// TwinCAT 3 PLC project REFLEX_3000_PLC
// ProgramVersion: 3.1.4023.0
// libraries:
//   Festo_HomingLibrary, * (Festo)
//   Festo_PtP_Base, * (Festo)
//   Festo_PtP_CiA402_ETC_CMMT_AS, * (Festo)
//   Festo_PtP_CiA402_ETC_CMMT_ST, * (Festo)
//   Tc2_EtherCAT, * (Beckhoff Automation GmbH)
//   Tc2_MC2, * (Beckhoff Automation GmbH)
//   Tc2_MC2_Drive, * (Beckhoff Automation GmbH)
//   Tc2_ModbusRTU, * (Beckhoff Automation GmbH)
//   Tc2_SerialCom, * (Beckhoff Automation GmbH)
//   Tc2_Standard, * (Beckhoff Automation GmbH)
//   Tc2_System, * (Beckhoff Automation GmbH)
//   Tc2_Utilities, * (Beckhoff Automation GmbH)
//   Tc3_EventLogger, * (Beckhoff Automation GmbH)
//   Tc3_Mc3Definitions, * (Beckhoff Automation GmbH)
//   Tc3_McCollisionAvoidance, * (Beckhoff Automation GmbH)
//   Tc3_McCoordinatedMotion, * (Beckhoff Automation GmbH)
//   Tc3_Module, * (Beckhoff Automation GmbH)
//   Util, * (System)
//   Tc3_XTS_Utility,3.1.2202.3,Beckhoff Automation GmbH
// project tree:
//   DUTs/ Running_Recipe.TcDUT
//   FB/Keyence_Laser/ FB_Keyence_Laser_Steuerung.TcPOU, ST_KeyenceLaser_Completion_Status.TcDUT, ST_KeyenceLaser_Count_Result_Data.TcDUT, ST_KeyenceLaser_ErrorStatus.TcDUT, ST_KeyenceLaser_Error_Codes.TcDUT, ST_KeyenceLaser_Function_Request.TcDUT, ST_KeyenceLaser_Function_Status.TcDUT, ST_KeyenceLaser_General_Request.TcDUT, ST_KeyenceLaser_Machine_Status.TcDUT, ST_KeyenceLaser_Operate_Parameter.TcDUT, ST_KeyenceLaser_Request_Completion_Clear.TcDUT, ST_KeyenceLaser_TwoD_Code_Read_Result.TcDUT
//   FB/Keyence_Laser/ST_Keyence/Input/ ST_KeyenceLaser_Block_Edit_Request_Completion_Status.TcDUT, ST_KeyenceLaser_Block_Edit_Request_Error_Status.TcDUT, ST_KeyenceLaser_Command_Request_Completion_Status.TcDUT, ST_KeyenceLaser_Command_Request_Error.TcDUT, ST_KeyenceLaser_Control_Status.TcDUT, ST_KeyenceLaser_Edit_Request_Completion_Status.TcDUT, ST_KeyenceLaser_Edit_Request_Error_Status.TcDUT, ST_KeyenceLaser_Function_Status_I.TcDUT, ST_KeyenceLaser_General_Request_Completion_Status.TcDUT, ST_KeyenceLaser_General_Request_Error_Status.TcDUT, ST_KeyenceLaser_General_Status.TcDUT, ST_KeyenceLaser_IO_Status.TcDUT, ST_KeyenceLaser_Operation_Request_Completion_Status.TcDUT, ST_KeyenceLaser_Operation_Request_Error_Status.TcDUT, ST_KeyenceLaser_Running_Status.TcDUT
//   FB/Keyence_Laser/ST_Keyence/Output/ ST_KeyenceLaser_Block_Edit_Request.TcDUT, ST_KeyenceLaser_Block_Edit_Request_Completion_Clear.TcDUT, ST_KeyenceLaser_Command_Request.TcDUT, ST_KeyenceLaser_Command_Request_Completion_Clear.TcDUT, ST_KeyenceLaser_Edit_Request.TcDUT, ST_KeyenceLaser_Edit_Request_Completion_Clear.TcDUT, ST_KeyenceLaser_Function_Request_I.TcDUT, ST_KeyenceLaser_General_Request_Completion_Clear.TcDUT, ST_KeyenceLaser_General_Request_I.TcDUT, ST_KeyenceLaser_Operating_Request.TcDUT, ST_KeyenceLaser_Operating_Request_Completion_Clear.TcDUT
//   FB/ OP10_ROBO_PNP.TcPOU, Servo_Conveyor_FB_OP90.TcPOU, Cylinder_Block.TcPOU, Cylinder_Block_FOR_OP130.TcPOU, Cylinder_Block_HOMING.TcPOU, FB_cycleTime.TcPOU, FB_SimClock.TcPOU, In_Range.TcPOU, Mode_Selection_Block1.TcPOU, OP10_ORING_PNP.TcPOU, OP140_LeakTesting.TcPOU, Pulse_1s.TcPOU, Servo_Conveyor_FB.TcPOU, TestSeq.TcPOU
//   FB/tool/ step_cycle_time.TcPOU, tool_changeover.TcPOU
//   POU1/ FB_Time_Stamp_Maddy.TcPOU, Axis_Position_Bias.TcPOU, MAIN.TcPOU, Recipe_Values.TcGVL, RFID.TcPOU
//   POUs/Programs/OP10/ Body_Singulation_Seq.TcPOU, OP10A_AUTO.TcPOU, OP10A_Camera_FB.TcPOU, OP10A_Conveyor_Prog.TcPOU, OP10A_OP10B_DRUM_FEEDER.TcPOU, OP10B_AUTO.TcPOU, OP10B_Camera_FB.TcPOU, OP10B_Conveyor_Prog.TcPOU, OP10_AUTO.TcPOU, OP10_Body_Camera_Seq.TcPOU, OP10_HMI_GVL.TcGVL, OP10_HOMING.TcPOU, OP10_MAIN.TcPOU, OP10_MANUAL.TcPOU, OP10_ROBO.TcPOU, OP10_SERVO.TcPOU, OP10_VARIABLE.TcGVL
//   POUs/Programs/OP120/ Bypass.TcDUT, OP120_AutoSequence.TcPOU, op120_camera_FB.TcPOU, OP120_Error.TcPOU, OP120_Feed_Conveyor.TcPOU, OP120_GVL.TcGVL, OP120_Initialization_Seq.TcPOU, OP120_IO_Tag_Link.TcGVL, OP120_LockInsert_AutoSequence.TcPOU, OP120_Main.TcPOU, OP120_Manual.TcPOU, OP120_Recipe.TcDUT, OP120_Robo_Byte_Mapping.TcPOU, OP120_Robo_Inputs.TcPOU, OP120_Sing_Auto_PRG.TcPOU
//   POUs/Programs/OP130/ op130_tool_change.TcPOU, OP130_AutoSequence.TcPOU, OP130_Error.TcPOU, OP130_GVL.TcGVL, OP130_Initialization_Seq.TcPOU, OP130_LH_Auto.TcPOU, OP130_Main.TcPOU, OP130_Manual.TcPOU, OP130_Recipe.TcDUT, OP130_RH_Auto.TcPOU, OP130_RH_Initialization_Seq.TcPOU
//   POUs/Programs/OP140/ op140_tool_change.TcPOU, Ateq_Comm_Prog.TcPOU, op140_ateq_fb.TcPOU, OP140_AutoSequence_1.TcPOU, OP140_AutoSequence_2.TcPOU, OP140_AutoSequence_3.TcPOU, OP140_Error.TcPOU, OP140_GVL.TcGVL, OP140_HMI_GVL.TcGVL, OP140_Initialization_Seq.TcPOU, OP140_Main.TcPOU, OP140_Manual.TcPOU
//   POUs/Programs/OP150/ OP150_B.TcPOU, OP150_Laser_FB.TcPOU, Rejection_Codes_Function.TcPOU, OP150_A.TcPOU, OP150_C.TcPOU, OP150_GVL.TcGVL, OP150_Main.TcPOU
//   POUs/Programs/OP20/ OP20_AUTOSEQUENCE.TcPOU, OP20_ERROR.TcPOU, OP20_GVL.TcGVL, OP20_Initialization_Seq.TcPOU, OP20_MAIN.TcPOU, OP20_MANUAL.TcPOU, OP20_Recipe.TcGVL
//   POUs/Programs/OP30/ OP30_Camera_FB.TcPOU, OP30_Conveyor_Cam_Seq.TcPOU, Camera_Job_Change.TcPOU, OP30_AUTOSEQUENCE.TcPOU, OP30_Error.TcPOU, OP30_GVL.TcGVL, OP30_HMI_TAGS.TcGVL, OP30_Initialize_Seq.TcPOU, OP30_MAIN.TcPOU, OP30_MANUAL.TcPOU, OP30_Recipe.TcGVL
//   POUs/Programs/OP40/ op40_toolchangeover.TcPOU, OP40_AUTOSEQUENCE.TcPOU, OP40_ERROR.TcPOU, OP40_GVL.TcGVL, OP40_Initialization_Seq.TcPOU, OP40_MAIN.TcPOU, OP40_MANUAL.TcPOU, OP40_Recipe.TcGVL
//   POUs/Programs/OP50/ OP50_Camera_FB.TcPOU, OP50_Conveyor_Cam_Seq.TcPOU, OP50_AUTOSEQUENCE.TcPOU, OP50_CONVEYOR.TcPOU, OP50_Error.TcPOU, OP50_GVL.TcGVL, OP50_HMI_GVL.TcGVL, OP50_Initialize_Seq.TcPOU, OP50_MAIN.TcPOU, OP50_MANUAL.TcPOU, OP50_Recipe.TcGVL
//   POUs/Programs/OP60/ op60_toolchangeover.TcPOU, OP60_AUTOSEQUENCE.TcPOU, OP60_ERROR.TcPOU, OP60_GVL.TcGVL, OP60_Initialization_Seq.TcPOU, OP60_MAIN.TcPOU, OP60_MANUAL.TcPOU, OP60_Recipe.TcGVL
//   POUs/Programs/OP70/ OP70_Camera_FB.TcPOU, OP70_Conveyor_Cam_Seq.TcPOU, OP70_AUTOSEQUENCE.TcPOU, OP70_CONVEYOR.TcPOU, OP70_Error.TcPOU, OP70_GVL.TcGVL, OP70_Initialize_Seq.TcPOU, OP70_MAIN.TcPOU, OP70_MANUAL.TcPOU, OP70_Recipe.TcGVL
//   POUs/Programs/OP80/ op80_toolchangeover.TcPOU, OP80_AUTOSEQUENCE.TcPOU, OP80_ERROR.TcPOU, OP80_GVL.TcGVL, OP80_HMI_GVL.TcGVL, OP80_Initialization_Seq.TcPOU, OP80_MAIN.TcPOU, OP80_MANUAL.TcPOU, OP80_Recipe.TcGVL
//   POUs/Programs/OP90/ OP90_Camera_Fb.TcPOU, OP90_AUTO.TcPOU, OP90_CAMERA.TcPOU, OP90_Conveyor_FBs.TcPOU, OP90_HMI_GVL.TcGVL, OP90_HOMING.TcPOU, OP90_MAIN.TcPOU, OP90_MANUAL.TcPOU, OP90_SERVO.TcPOU, OP90_VARIABLE.TcGVL
//   POUs/Programs/XTS/ Fb_MoverSequence.TcPOU, HMI_GVL.TcGVL, MAIN_1.TcPOU, PRG_XTS_Sequence.TcPOU, XTS_GVL.TcGVL
//   / Robot_Comm_Task.TcTTO, PlcTask.TcTTO, RecipeManager.TcRMO (not stored)
//   DUTs/OP10/ OP10_GRP_CONTRL.TcDUT, OP10_GRP_STATUS.TcDUT, OP10_ORNG_CYL_DLY.TcDUT, OP10_ORNG_CYL_IP.TcDUT, OP10_ORNG_CYL_OP.TcDUT, OP10_ROBO_CNTRL.TcDUT, OP10_ROBO_STUS.TcDUT
//   DUTs/XTS/ STATION_DONE.TcDUT
//   FB/Axis/ ENUM_Axis.TcDUT, FB_Axis.TcPOU, FB_Axis_FESTO.TcPOU, OP10_SERVO_LIMIT.TcDUT, OP90_SERVO_LIMIT.TcDUT, Servo_Control.TcDUT, stManualModeAxis.TcDUT
//   FB/Cognex_Camera/ Acquisition_control.TcDUT, Acquisition_status.TcDUT, FB_Cognex_ProfiNET_1.TcPOU, Inspection_control.TcDUT, Inspection_status.TcDUT, UNION_64Byte.TcDUT
//   FB/FB/FB/ ATEQ_LEAK.TcPOU
//   FB/RFID/ FB_RFID.TcPOU, Head1.TcDUT, HeadData.TcDUT, Memory.TcDUT, UNION_RFID.TcDUT
//   FB/Robot/ E_State_RobotGeneral.TcDUT, FB_Robot.TcPOU
//   FB/Scanner/ Acquisition_Control_Scanner.TcDUT, Acquisition_Status_Scanner.TcDUT, Result_Control_Scanner.TcDUT, Result_Data_Register.TcDUT, Result_Status.TcDUT, Scanner.TcPOU
//   FB/Schunk/ ENUM_Schunk.TcDUT, FB_Schunk.TcPOU, FC_Real_Convert.TcPOU, iSchunkProcessData.TcDUT, oSchunkProcessData.TcDUT, stManualModeAxis_1.TcDUT, UNION_iSchunkProcessData.TcDUT, UNION_oSchunkProcessData.TcDUT, UNION_REAL.TcDUT
//   GVLs/ E_EcCommState.TcDUT, GVL.TcGVL, RayPRO_Variables.TcGVL, SerialComm.TcGVL, ST_SlaveState.TcDUT, ST_SlaveStateInfo.TcDUT (not stored)
//   GVLs/XTS/ GVL_XTS.TcGVL
//   POUs/ Error.TcPOU
//   POUs/GENERAL/ Robot_232_Comm_Prgrm.TcPOU, EtherCatDiag.TcPOU, GENERAL_VARIABLE.TcGVL, IO_Diag.TcPOU, MODE_SELECTION.TcPOU
//   POUs/IO/ OP120_JB_IO.TcPOU, OP160_MASTER4_IO.TcPOU, OP160_MP_IO.TcPOU, OP90_JB_IO.TcPOU, OP90_MASTER3_IO.TcPOU, OP90_MP_IO.TcPOU
//   POUs/IO_GVLs/ Master3_IO.TcGVL, Master4_IO.TcGVL, OP120_JB.TcGVL, OP160_MP.TcGVL, OP90_JB.TcGVL, OP90_MP.TcGVL, SAFETY_IOs.TcGVL
//   POUs/IO_Mapping_OP10JB/ IO_OP10A_10B_JB.TcPOU, IO_OP10_JB_IO.TcGVL
//   POUs/IO_mapping_OP10MP/ IO_OP10_MP.TcGVL, IO_OP10_PANEL.TcPOU
//   POUs/OP10_Profinet_IO/ Master1_IO.TcGVL, Master1_IO_Map.TcPOU, MASTER2_IO.TcGVL, MASTER2_IO_Map.TcPOU
//   POUs/Programs/ Error_GVL.TcGVL
//   POUs/Programs/offline testing/ cylinder_2_pos.TcPOU, cylinder_3_pos.TcPOU, Cylinder_Block_v1.TcPOU, cylinder_validation_st.TcPOU, offline_fb.TcPOU, offline_main.TcPOU, POU_1.TcPOU, servo.TcPOU, servo_validation.TcPOU
//   POUs/Programs/OP10A_Bowl/ Bowl_Control.TcPOU
//   POUs/Programs/OP110/ OP110_AUTOSEQUENCE.TcPOU, OP110_ERROR.TcPOU, OP110_GVL.TcGVL, OP110_HMI_GVL.TcGVL, OP110_Initialization_Seq.TcPOU, OP110_MAIN.TcPOU, OP110_MANUAL.TcPOU, OP110_Recipe.TcGVL
//   POUs/Programs/OP160/ OP160_AutoSequence.TcPOU, OP160_Error.TcPOU, OP160_GVL.TcGVL, OP160_Initialization_Seq.TcPOU, OP160_IO_Tag_Link.TcGVL, OP160_Main.TcPOU, OP160_Manual.TcPOU, OP160_QCPlace_AutoSequence.TcPOU, OP160_Recipe.TcDUT, OP160_RFID.TcPOU, OP160_Robo_Byte_Mapping.TcPOU, OP160_Robo_Inputs.TcPOU

CONFIGURATION REFLEX_3000_PLC
    RESOURCE PLC ON TwinCAT3
        TASK Robot_Comm_Task(INTERVAL := T#1ms, PRIORITY := 19);
        TASK PlcTask(INTERVAL := T#10ms, PRIORITY := 20);
        PROGRAM Robot_232_Comm_Prgrm WITH Robot_Comm_Task : Robot_232_Comm_Prgrm;
        PROGRAM MAIN WITH PlcTask : MAIN;
    END_RESOURCE
END_CONFIGURATION

// ---- DUTs/Running_Recipe.TcDUT
TYPE Running_Recipe :
STRUCT
//General
	Model_Dia					: STRING[80];
	Part_Number					: STRING[80];
	Body_Conductivity			: BOOL;
	Comp_Per_Bag 				: INT;
		
//OP10	
	OP10_Cam_Prog_Num			: INT;
	OP10_Robot_Prog_Num			: INT;
	OP10_Gripper_Pos			: REAL;

//OP20
	OP20_Vert_Ser_Pos			: REAL;
	OP20_Oiling_Time			: INT;
	
OP20_Oiling_Range				: REAL;

//OP30
	OP30_Cam_Prog_Num			: INT;
	OP30_Grip_Wrk_Pos			: REAL;
	OP30_Vert_Ser_Pick_Pos		: REAL;
	OP30_Vert_Ser_Place_Pos		: REAL;	
	OP30_Hori_Ser_Pick_Pos		: REAL;
	OP30_Hori_Ser_Place_Pos		: REAL;		

//OP40
	OP40_Vert_Ser_Pos			: REAL;
	OP40_LVDT_Chck_Value		: REAL;

//OP40_LVDT_Tolerance				: REAL;

//OP50
	OP50_Cam_Prog_Num			: INT;
	OP50_Vert_Ser_Pick_Pos		: REAL;
	OP50_Vert_Ser_Place_Pos		: REAL;	
	OP50_Hori_Ser_Pick_Pos		: REAL;
	OP50_Hori_Ser_Place_Pos		: REAL;		

//OP60
	OP60_Vert_Ser_Pos			: REAL;
	OP60_LVDT_Chck_Value		: REAL;

//OP60_LVDT_Tolerance				: REAL;

//OP70
	OP70_Cam_Prog_Num			: INT;
	OP70_Grip_Wrk_Pos			: REAL;
	OP70_Vert_Ser_Pick_Pos		: REAL;
	OP70_Vert_Ser_Place_Pos		: REAL;	
	OP70_Hori_Ser_Pick_Pos		: REAL;
	OP70_Hori_Ser_Place_Pos		: REAL;		


//OP80
	OP80_Vert_Ser_Pos			: REAL;
	OP80_LVDT_Chck_Value		: REAL;

//OP80_LVDT_Tolerance				: REAL;

//OP90
	OP90_Cam_Prog_Num			: INT;
	OP90_Vert_Ser_Pick_Pos		: REAL;
	OP90_Vert_Ser_Place_Pos		: REAL;	
	OP90_Hori_Ser_Pick_Pos		: REAL;
	OP90_Hori_Ser_Place_Pos		: REAL;	

//OP110
	OP110_Vert_Ser_Pos			: REAL;
	OP110_Oiling_Time			: INT;
	
OP110_Oiling_Range				: REAL;

//OP120
	OP120_Cam_Prog_Num			: INT;
                            	
//OP130                     	
	OP130_Trq_value				: REAL;
	OP130_Vert_Ser_Pos			: REAL;
	                        	
//OP140                     	
	OP140_Vert_Ser_Pos			: REAL;
	                        	
OP140_Wiping_Cycle				: INT;
OP140_NOK_Retry_Cycle			: INT;
                            	
//OP150-A                   	
	OP150A_Cam_Prog_Num			: INT;
	                        	
//OP150-B                   	
	OP150B_Lsr_Mrk_Job_num		: INT;
	
//OP160
	OP160_Robo_Prog_Num			: INT;	
END_STRUCT
END_TYPE

// ---- FB/Keyence_Laser/ST_KeyenceLaser_Completion_Status.TcDUT
TYPE ST_KeyenceLaser_Completion_Status :
STRUCT
Marking_Complete				: BIT ;
Guide_Laser_Complete			: BIT ;
Laser_Stop_Complete				: BIT ;
Error_Clear_Complete			: BIT ;
TWODC_Read_Complete				: BIT ;
Reserve_15						: BIT ;
Reserve_16						: BIT ;
Reserve_17						: BIT ;
//
PROGRAM_Edit_Complete			: BIT ;
Reserve_18						: BIT ;
Reserve_19						: BIT ;
Reserve_20						: BIT ;
Reserve_21						: BIT ;
Reserve_22						: BIT ;
Reserve_23						: BIT ;
Reserve_24						: BIT ;
//
PROGRAM_Change_Complete			: BIT ;
Rank_Change_Complete			: BIT ;
Counter_No_Complete				: BIT ;
Counter_Value_Complete			: BIT ;
Counter_Up_Complete				: BIT ;
Counter_Down_Complete			: BIT ;
Counter_Reset_Complete			: BIT ;
Reserve_25						: BIT ;
//
ReserveByte_2					: Byte ;
//
Setting_STRING_Read_Complete	: BIT ;
Marked_STRING_Read_Complete		: BIT ;
STRING_Change_Complete			: BIT ;
Reserve_26						: BIT ;
Reserve_27						: BIT ;
Reserve_28						: BIT ;
Reserve_29						: BIT ;
Reserve_30						: BIT ;
//
ReserveWord_2a					: BYTE ;
//
ReserveWord_2b					: BYTE ;
//
Command_Send_Complete			: BIT ;
Reserve_31						: BIT ;
Reserve_32						: BIT ;
Reserve_33						: BIT ;
Reserve_34						: BIT ;
Reserve_35						: BIT ;
Reserve_36						: BIT ;
Reserve_37						: BIT ;
END_STRUCT
END_TYPE

// ---- FB/Keyence_Laser/ST_KeyenceLaser_Count_Result_Data.TcDUT
TYPE ST_KeyenceLaser_Count_Result_Data :
STRUCT
END_STRUCT
END_TYPE

// ---- FB/Keyence_Laser/ST_KeyenceLaser_ErrorStatus.TcDUT
TYPE ST_KeyenceLaser_ErrorStatus :
STRUCT
Start_Marking_Request_Error			: BIT ;
Guide_Laser_Request_Error			: BIT ;
Stop_Marking_Request_Error			: BIT ;
Error_Clear_Request_Error			: BIT ;
TwoDC_Read_Request_Error			: BIT ;//2DC_Read_Request_Error
Reserve_38							: BIT ;
Reserve_39							: BIT ;
Reserve_40							: BIT ;
//
PROGRAM_Edit_Error					: BIT ;
Reserve_41							: BIT ;
Reserve_42							: BIT ;
Reserve_43							: BIT ;
Reserve_44							: BIT ;
Reserve_45							: BIT ;
Reserve_46							: BIT ;
Reserve_47							: BIT ;
//
PROGRAM_Change_Request_Error		: BIT ;
Rank_Change_Request_Error			: BIT ;
Counter_No_Change_Request_Error		: BIT ;
Counter_Value_Change_Request_Error	: BIT ;
Counter_Up_Request_Error			: BIT ;
Counter_Down_Request_Error			: BIT ;
Counter_Reset_Request_Error			: BIT ;
Reserve_48							: BIT ;
//
ReserveByte_3						: Byte ;
//
Setting_STRING_Read_Request_Error	: BIT ;
Marked_STRING_Read_Request_Error	: BIT ;
STRING_Change_Request_Error			: BIT ;
Reserve_49							: BIT ;
Reserve_50							: BIT ;
Reserve_51							: BIT ;
Reserve_52							: BIT ;
Reserve_53							: BIT ;
//
ReserveWord_3a						: Byte ;
//
ReserveWord_3b						: Byte ;
//
Command_Send_Request_Error			: BIT ;
Reserve_54							: BIT ;
Reserve_55							: BIT ;
Reserve_56							: BIT ;
Reserve_57							: BIT ;
Reserve_58							: BIT ;
Reserve_59							: BIT ;
Reserve_60							: BIT ;
END_STRUCT
END_TYPE

// ---- FB/Keyence_Laser/ST_KeyenceLaser_Error_Codes.TcDUT
TYPE ST_KeyenceLaser_Error_Codes :
STRUCT
Error_Code_1				: WORD ;
Error_Code_2				: WORD ;
Command_Send_Error_Status	: WORD ;
ReserveWord_4				: WORD ;
END_STRUCT
END_TYPE

// ---- FB/Keyence_Laser/ST_KeyenceLaser_Function_Request.TcDUT
TYPE ST_KeyenceLaser_Function_Request :
STRUCT
Trigger_Lock_Request	: BIT ;
Operation_Stop_Request	: BIT ;
Laser_Stop_Request		: BIT ;
Date_Hold_Request		: BIT ;
A_Reserve_24			: BIT ;
A_Reserve_25			: BIT ;
A_Reserve_26			: BIT ;
A_Reserve_27			: BIT ;
//
A_ReserveByte_4			: Byte ;
A_ReserveWord1			: Word ;
END_STRUCT
END_TYPE

// ---- FB/Keyence_Laser/ST_KeyenceLaser_Function_Status.TcDUT
TYPE ST_KeyenceLaser_Function_Status :
STRUCT
Trigger_Lock_Status				: BIT ;
Operation_Stop_Status			: BIT ;
Laser_Control_Status			: BIT ;
DATE_Hold_Status				: BIT ;
Reserve_10						: BIT ;
Reserve_11						: BIT ;
Reserve_12						: BIT ;
Reserve_13						: BIT ;
//
DATE_Attach_Status				: BIT ;
Counter_End1_Status				: BIT ;
Counter_End2_Status				: BIT ;
Counter_End3_Status				: BIT ;
Counter_End4_Status				: BIT ;
Mark_Check_TwoDC_Read_OK_Status	: BIT ;//Mark_Check_2DC_Read_OK_Status
Mark_Check_TwoDC_Read_NG_Status	: BIT ;//Mark_Check_2DC_Read_NG_Status
Reserve_14						: BIT ;
//
ReserveWord_1					: WORD ;
END_STRUCT
END_TYPE

// ---- FB/Keyence_Laser/ST_KeyenceLaser_General_Request.TcDUT
TYPE ST_KeyenceLaser_General_Request :
STRUCT
Start_Marking_Request			: BIT ;
Guide_Laser_Request				: BIT ;
Stop_Marking_Request			: BIT ;
Error_Clear_Request				: BIT ;
TwoD_C_Read_Request				: BIT ;//2DC_Read_Request
A_Reserve_1						: BIT ;
A_Reserve_2						: BIT ;
A_Reserve_3						: BIT ;
//
Program_Edit_Start_Request		: BIT ;
A_Reserve_4						: BIT ;
A_Reserve_5						: BIT ;
A_Reserve_6						: BIT ;
A_Reserve_7						: BIT ;
A_Reserve_8						: BIT ;
A_Reserve_9						: BIT ;
A_Reserve_10					: BIT ;
//
Program_Change_Request			: BIT ;
Rank_Change_Request				: BIT ;
Counter_No_Change_Request		: BIT ;
Counter_Value_Change_Request	: BIT ;
Counter_Up_Request				: BIT ;
Counter_Down_Request			: BIT ;
Counter_Reset_Request			: BIT ;
A_Reserve_11					: BIT ;
//
A_ReserveByte_1					: BYTE ;
//
A_ReserveByte_2					: BYTE ;
//
Setting_String_Read_Request		: BIT ;
Marked_String_Read_Request		: BIT ;
STRING_Change_Request			: BIT ;
A_Reserve_12					: BIT ;
A_Reserve_13					: BIT ;
A_Reserve_14					: BIT ;
A_Reserve_15					: BIT ;
A_Reserve_16					: BIT ;
//
A_ReserveByte_3					: Byte ;
//
Command_Send_Request			: BIT ;
A_Reserve_17					: BIT ;
A_Reserve_18					: BIT ;
A_Reserve_19					: BIT ;
A_Reserve_20					: BIT ;
A_Reserve_21					: BIT ;
A_Reserve_22					: BIT ;
A_Reserve_23					: BIT ;
END_STRUCT
END_TYPE

// ---- FB/Keyence_Laser/ST_KeyenceLaser_Machine_Status.TcDUT
TYPE ST_KeyenceLaser_Machine_Status :
STRUCT
Ready_Status						: BIT ;
Error_Status						: BIT ;
Warning_Status						: BIT ;
Error_Warning_Status				: BIT ;
Shutter_Status						: BIT ;
Network_Status						: BIT ;
Reserve_1							: BIT ;
Reserve_2							: BIT ;
//
Laser_Emitted_Status				: BIT ;
Shutter_Control_Status				: BIT ;
Remote_Interlock_Status				: BIT ;
Contacter_Status					: BIT ;
Reserve_3							: BIT ;
Reserve_4							: BIT ;
Reserve_5							: BIT ;
Reserve_6							: BIT ;
//
Busy_Status							: BIT ;
Marking_Busy_Status					: BIT ;
Guide_Laser_Busy_Status				: BIT ;
PROGRAM_Change_Busy_Status			: BIT ;
Communication_Prioirty_Error_Status	: BIT ;
PROGRAM_Edit_Busy_Status			: BIT ;
Mark_Check_TwoDC_Read_Busy_Status	: BIT ;//Mark_Check_/2DC_Read_Busy_Status
Reserve_7							: BIT ;
//
ReserveByte_1						: BYTE ;
END_STRUCT
END_TYPE

// ---- FB/Keyence_Laser/ST_KeyenceLaser_Operate_Parameter.TcDUT
TYPE ST_KeyenceLaser_Operate_Parameter :
STRUCT
PROGRAM_No_Status		: WORD ;
Counter_No_Status		: WORD ;
Counter_Value_Status	: DWORD ;
Rank_Value_Status		: WORD ;
ReserveWord_5			: WORD ;
ReserveDWord_1			: DWORD ;
END_STRUCT
END_TYPE

// ---- FB/Keyence_Laser/ST_KeyenceLaser_Request_Completion_Clear.TcDUT
TYPE ST_KeyenceLaser_Request_Completion_Clear :
STRUCT
Marking_Complete_BIT_Clear					: BIT ;
Guide_Laser_Complete_Bit_Clear				: BIT ;
Stop_Marking_Complete_Bit_Clear				: BIT ;
Error_Clear_Complete_Bit_Clear				: BIT ;
TwoDC_Read_Complete_Bit_Clear				: BIT ;//2DC_Read_Complete_Bit_Clear	
A_Reserve_28								: BIT ;
A_Reserve_29								: BIT ;
A_Reserve_30								: BIT ;
//
Program_Edit_Complete_Bit_Clear				: BIT ;
A_Reserve_31								: BIT ;
A_Reserve_32								: BIT ;
A_Reserve_33								: BIT ;
A_Reserve_34								: BIT ;
A_Reserve_35								: BIT ;
A_Reserve_36								: BIT ;
A_Reserve_37								: BIT ;
//
Program_Change_Complete_Bit_Clear			: BIT ;
Rank_Change_Complete_Bit_Clear				: BIT ;
Counter_No_Change_Complete_Bit_Clear		: BIT ;
Counter_Value_Change_Complete_Bit_Clear		: BIT ;
Count_Up_Complete_Bit_Clear					: BIT ;
Count_Down_Complete_Bit_Clear				: BIT ;
Counter_Reset_Complete_Bit_Clear			: BIT ;
A_Reserve_38								: BIT ;
//
A_ReserveByte_5								: Byte ;
//
Setting_String_Read_Complete_Bit_Clear		: BIT ;
Marked_String_Read_Complete_Bit_Clear		: BIT ;
String_Change_Complete_Bit_Clear			: BIT ;
A_Reserve_39								: BIT ;
A_Reserve_40								: BIT ;
A_Reserve_41								: BIT ;
A_Reserve_42								: BIT ;
A_Reserve_43								: BIT ;
//
A_ReserveByte_6								: Byte ;
//
A_ReserveByte_7								: Byte ;
//
Command_Send_Complete_Bit_Clear				: BIT ;
A_Reserve_44								: BIT ;
A_Reserve_45								: BIT ;
A_Reserve_46								: BIT ;
A_Reserve_47								: BIT ;
A_Reserve_48								: BIT ;
A_Reserve_49								: BIT ;
A_Reserve_50								: BIT ;
END_STRUCT
END_TYPE

// ---- FB/Keyence_Laser/ST_KeyenceLaser_TwoD_Code_Read_Result.TcDUT

TYPE ST_KeyenceLaser_TwoD_Code_Read_Result :
STRUCT
Marking_Check_Score_TwoDC_Read_Grade_Status		: WORD ;
Check_Count_Status								: WORD ;
ReserveDWord_2									: DWORD ;
END_STRUCT
END_TYPE

// ---- FB/Keyence_Laser/ST_Keyence/Input/ST_KeyenceLaser_Block_Edit_Request_Completion_Status.TcDUT
TYPE ST_KeyenceLaser_Block_Edit_Request_Completion_Status :
STRUCT
Character_String_Setting_Read_Complete			: BIT;
Character_String_Printed_Read_Complete			: BIT;
Character_String_Change_Complete				: BIT;
Reserve_0										: BIT;
Reserve_1										: BIT;
Reserve_2										: BIT;
Reserve_3										: BIT;
Reserve_4										: BIT;
END_STRUCT
END_TYPE

// ---- FB/Keyence_Laser/ST_Keyence/Input/ST_KeyenceLaser_Block_Edit_Request_Error_Status.TcDUT
TYPE ST_KeyenceLaser_Block_Edit_Request_Error_Status :
STRUCT
Character_String_Setting_Read_Error				: BIT;
Character_String_Printed_Read_Error				: BIT;
Character_String_Change_Error					: BIT;
Reserve_0										: BIT;
Reserve_1										: BIT;
Reserve_2										: BIT;
Reserve_3										: BIT;
Reserve_4										: BIT;
END_STRUCT
END_TYPE

// ---- FB/Keyence_Laser/ST_Keyence/Input/ST_KeyenceLaser_Command_Request_Completion_Status.TcDUT
TYPE ST_KeyenceLaser_Command_Request_Completion_Status :
STRUCT
Command_Request_Complete			: BIT;
Reserve_0							: BIT;
Reserve_1							: BIT;
Reserve_2							: BIT;
Reserve_3							: BIT;
Reserve_4							: BIT;
Reserve_5							: BIT;
Reserve_6							: BIT;
END_STRUCT
END_TYPE

// ---- FB/Keyence_Laser/ST_Keyence/Input/ST_KeyenceLaser_Command_Request_Error.TcDUT
TYPE ST_KeyenceLaser_Command_Request_Error :
STRUCT
Command_Request_Error				: BIT;
Reserve_0							: BIT;
Reserve_1							: BIT;
Reserve_2							: BIT;
Reserve_3							: BIT;
Reserve_4							: BIT;
Reserve_5							: BIT;
Reserve_6							: BIT;
END_STRUCT
END_TYPE

// ---- FB/Keyence_Laser/ST_Keyence/Input/ST_KeyenceLaser_Control_Status.TcDUT
TYPE ST_KeyenceLaser_Control_Status :
STRUCT
Data_Hold							: BIT;
Counter_End_1						: BIT;
Counter_End_2						: BIT;
Counter_End_3						: BIT;
Counter_End_4						: BIT;
TwoD_Code_Read_OK					: BIT;
TwoD_Code_Read_NG					: BIT;
Marking_Complete_1					: BIT;
END_STRUCT
END_TYPE

// ---- FB/Keyence_Laser/ST_Keyence/Input/ST_KeyenceLaser_Edit_Request_Completion_Status.TcDUT
TYPE ST_KeyenceLaser_Edit_Request_Completion_Status :
STRUCT
Edit_Complete		: BIT;
Reserve_0			: BIT;
Reserve_1			: BIT;
Reserve_2			: BIT;
Reserve_3			: BIT;
Reserve_4			: BIT;
Reserve_5			: BIT;
Reserve_6			: BIT;
END_STRUCT
END_TYPE

// ---- FB/Keyence_Laser/ST_Keyence/Input/ST_KeyenceLaser_Edit_Request_Error_Status.TcDUT
TYPE ST_KeyenceLaser_Edit_Request_Error_Status :
STRUCT
Edit_Error			: BIT;
Reserve_0			: BIT;
Reserve_1			: BIT;
Reserve_2			: BIT;
Reserve_3			: BIT;
Reserve_4			: BIT;
Reserve_5			: BIT;
Reserve_6			: BIT;
END_STRUCT
END_TYPE

// ---- FB/Keyence_Laser/ST_Keyence/Input/ST_KeyenceLaser_Function_Status_I.TcDUT
TYPE ST_KeyenceLaser_Function_Status_I :
STRUCT
Trigger_Inhibit_Function_Status							: BIT;
Machinery_Operation_Mode_Disable_Function_Status		: BIT;
Marking_Laser_Control_Function_Status					: BIT;
Data_Hold_Function_Status								: BIT;
Reserve_0												: BIT;
Reserve_1												: BIT;
Reserve_2												: BIT;
Reserve_3												: BIT;
END_STRUCT
END_TYPE

// ---- FB/Keyence_Laser/ST_Keyence/Input/ST_KeyenceLaser_General_Request_Completion_Status.TcDUT
TYPE ST_KeyenceLaser_General_Request_Completion_Status :
STRUCT
Marking_Complete_2		: BIT;
Guide_Print_Complete	: BIT;
Print_Stop_Complete		: BIT;
Error_Clear_Complete	: BIT;
TwoDC_Read_Complete		: BIT;
Reserve_4				: BIT;
Reserve_5				: BIT;
Reserve_6				: BIT;
END_STRUCT
END_TYPE

// ---- FB/Keyence_Laser/ST_Keyence/Input/ST_KeyenceLaser_General_Request_Error_Status.TcDUT
TYPE ST_KeyenceLaser_General_Request_Error_Status :
STRUCT
Print_Error				: BIT;
Guide_Print_Error		: BIT;
Print_Stop_Error		: BIT;
Error_Clear_Error		: BIT;
TwoDC_Read_Error		: BIT;
Reserve_0				: BIT;
Reserve_1				: BIT;
Reserve_2				: BIT;
END_STRUCT
END_TYPE

// ---- FB/Keyence_Laser/ST_Keyence/Input/ST_KeyenceLaser_General_Status.TcDUT
TYPE ST_KeyenceLaser_General_Status :
STRUCT
Ready_Status						: BIT;
Error_Status						: BIT;
Warning_Status						: BIT;
Notice_Status						: BIT;
Shutter_Status						: BIT;
StartUp_Status						: BIT;
Program_Change_Ready				: BIT;
Reserve								: BIT;
END_STRUCT
END_TYPE

// ---- FB/Keyence_Laser/ST_Keyence/Input/ST_KeyenceLaser_IO_Status.TcDUT
TYPE ST_KeyenceLaser_IO_Status :
STRUCT
Laser_Emit_Status					: BIT;
Shutter_Control_Status				: BIT;
Remote_Interlock_Status				: BIT;
Contactor_Status					: BIT;
Reserve_0							: BIT;
Reserve_1							: BIT;
Reserve_2							: BIT;
Reserve_3							: BIT;
END_STRUCT
END_TYPE

// ---- FB/Keyence_Laser/ST_Keyence/Input/ST_KeyenceLaser_Operation_Request_Completion_Status.TcDUT
TYPE ST_KeyenceLaser_Operation_Request_Completion_Status :
STRUCT
Program_Change_Complete				: BIT;
Ranke_Value_Change_Complete			: BIT;
Counter_Number_Change_Complete		: BIT;
Counter_Value_Change_Complete		: BIT;
Counter_Up_Complete					: BIT;
Counter_Down_Complete				: BIT;
Counter_Reset_Complete				: BIT;
Reserve								: BIT;
END_STRUCT
END_TYPE

// ---- FB/Keyence_Laser/ST_Keyence/Input/ST_KeyenceLaser_Operation_Request_Error_Status.TcDUT
TYPE ST_KeyenceLaser_Operation_Request_Error_Status :
STRUCT
Program_Change_error				: BIT;
Rank_Value_Change					: BIT;
Counter_Number_Change_Error			: BIT;
Counter_Value_Change_Error			: BIT;
Counter_Up_Error					: BIT;
Counter_Down_Error					: BIT;
Counter_Reset_Error					: BIT;
Reserve								: BIT;
END_STRUCT
END_TYPE

// ---- FB/Keyence_Laser/ST_Keyence/Input/ST_KeyenceLaser_Running_Status.TcDUT
TYPE ST_KeyenceLaser_Running_Status :
STRUCT
Busy_Status							: BIT;
Print_Busy_Status					: BIT;
Guide_Print_Busy_Status				: BIT;
Program_Change_Busy_Status			: BIT;
Lock_Busy_Status					: BIT;
Edit_Busy_Status					: BIT;
TwoDC_Read_Busy_Status				: BIT;
Reserve								: BIT;
END_STRUCT
END_TYPE

// ---- FB/Keyence_Laser/ST_Keyence/Output/ST_KeyenceLaser_Block_Edit_Request.TcDUT
TYPE ST_KeyenceLaser_Block_Edit_Request :
STRUCT
Character_String_Setting_Read_Request		: BIT;
Character_String_Printed_Read_Request		: BIT;
Character_String_Change_Request				: BIT;
Reserve_0									: BIT;
Reserve_1									: BIT;
Reserve_2									: BIT;
Reserve_3									: BIT;
Reserve_4									: BIT;
END_STRUCT
END_TYPE

// ---- FB/Keyence_Laser/ST_Keyence/Output/ST_KeyenceLaser_Block_Edit_Request_Completion_Clear.TcDUT
TYPE ST_KeyenceLaser_Block_Edit_Request_Completion_Clear :
STRUCT
Character_String_Setting_Read_Complete_Clear		: BIT;
Character_String_Printed_Read_Complete_Clear		: BIT;
Character_String_Change_Complete_Clear				: BIT;
Reserve_0											: BIT;
Reserve_1											: BIT;
Reserve_2											: BIT;
Reserve_3											: BIT;
Reserve_4											: BIT;
END_STRUCT
END_TYPE

// ---- FB/Keyence_Laser/ST_Keyence/Output/ST_KeyenceLaser_Command_Request.TcDUT
TYPE ST_KeyenceLaser_Command_Request :
STRUCT
Command_Request		: BIT;
Reserve_0			: BIT;
Reserve_1			: BIT;
Reserve_2			: BIT;
Reserve_3			: BIT;
Reserve_4			: BIT;
Reserve_5			: BIT;
Reserve_6			: BIT;
END_STRUCT
END_TYPE

// ---- FB/Keyence_Laser/ST_Keyence/Output/ST_KeyenceLaser_Command_Request_Completion_Clear.TcDUT
TYPE ST_KeyenceLaser_Command_Request_Completion_Clear :
STRUCT
Command_Request_Complete_Clear		: BIT;
Reserve_0							: BIT;
Reserve_1							: BIT;
Reserve_2							: BIT;
Reserve_3							: BIT;
Reserve_4							: BIT;
Reserve_5							: BIT;
Reserve_6							: BIT;
END_STRUCT
END_TYPE

// ---- FB/Keyence_Laser/ST_Keyence/Output/ST_KeyenceLaser_Edit_Request.TcDUT
TYPE ST_KeyenceLaser_Edit_Request :
STRUCT
Edit_Start_Request			: BIT;
Reserve_0					: BIT;
Reserve_1					: BIT;
Reserve_2					: BIT;
Reserve_3					: BIT;
Reserve_4					: BIT;
Reserve_5					: BIT;
Reserve_6					: BIT;
END_STRUCT
END_TYPE

// ---- FB/Keyence_Laser/ST_Keyence/Output/ST_KeyenceLaser_Edit_Request_Completion_Clear.TcDUT
TYPE ST_KeyenceLaser_Edit_Request_Completion_Clear :
STRUCT
Edit_Complete_Clear			: BIT;
Reserve_0					: BIT;
Reserve_1					: BIT;
Reserve_2					: BIT;
Reserve_3					: BIT;
Reserve_4					: BIT;
Reserve_5					: BIT;
Reserve_6					: BIT;
END_STRUCT
END_TYPE

// ---- FB/Keyence_Laser/ST_Keyence/Output/ST_KeyenceLaser_Function_Request_I.TcDUT
TYPE ST_KeyenceLaser_Function_Request_I :
STRUCT
Trigger_Inhibit_Function_Request							: BIT;
Machinery_Operation_Mode_Disable_Function_Request			: BIT;
Marking_Laser_Control_Function_Request						: BIT;
Date_Hold_Function_Request									: BIT;
Reserve_0													: BIT;
Reserve_1													: BIT;
Reserve_2													: BIT;
Reserve_3													: BIT;
END_STRUCT
END_TYPE

// ---- FB/Keyence_Laser/ST_Keyence/Output/ST_KeyenceLaser_General_Request_Completion_Clear.TcDUT
TYPE ST_KeyenceLaser_General_Request_Completion_Clear :
STRUCT
Print_Complete_Clear						: BIT;
Guide_Print_Complete_Clear					: BIT;
Print_Stop_Complete_Clear					: BIT;
Error_Clear_Complete_Clear					: BIT;
TwoD_Code_Read_Complete_Clear				: BIT;
Reserve_0									: BIT;
Reserve_1									: BIT;
Reserve_2									: BIT;
END_STRUCT
END_TYPE

// ---- FB/Keyence_Laser/ST_Keyence/Output/ST_KeyenceLaser_General_Request_I.TcDUT
TYPE ST_KeyenceLaser_General_Request_I :
STRUCT
Print_Start_Request				: BIT;
Guide_Print_Start_Request		: BIT;
Print_Stop_Request				: BIT;
Error_Clear_Request				: BIT;
TwoDC_Code_Read_Request			: BIT;
Reserve_0						: BIT;
Reserve_1						: BIT;
Reserve_2						: BIT;
END_STRUCT
END_TYPE

// ---- FB/Keyence_Laser/ST_Keyence/Output/ST_KeyenceLaser_Operating_Request.TcDUT
TYPE ST_KeyenceLaser_Operating_Request :
STRUCT
Program_Change_Request			: BIT;
Rank_Value_Change_Request		: BIT;
Counter_Number_Change_Request	: BIT;
Counter_Value_Change_Request	: BIT;
Counter_Up_Request				: BIT;
Counter_Down_Request			: BIT;
Counter_Reset_Request			: BIT;
Reserve							: BIT;
END_STRUCT
END_TYPE

// ---- FB/Keyence_Laser/ST_Keyence/Output/ST_KeyenceLaser_Operating_Request_Completion_Clear.TcDUT
TYPE ST_KeyenceLaser_Operating_Request_Completion_Clear :
STRUCT
Program_Change_Complete_Clear			: BIT;
Rank_Value_Change_Complete_Clear		: BIT;
Counter_Number_Change_Complete_Clear	: BIT;
Counter_Value_Change_Complete_Clear		: BIT;
Counter_Up_Complete_Clear				: BIT;
Counter_Down_Complete_Clear				: BIT;
Counter_Reset_Complete_Clear			: BIT;
Reserve									: BIT;
END_STRUCT
END_TYPE

// ---- POUs/Programs/OP120/Bypass.TcDUT
TYPE Bypass :
STRUCT
OP120_Bypass_1:		BOOL;
OP120_Bypass_2:		BOOL;
OP120_Bypass_3:		BOOL;
OP120_Bypass_4:		BOOL;
OP120_Bypass_5:		BOOL;
OP120_Bypass_6:		Bool;
OP120_Bypass_7:		Bool;
OP120_Bypass_8:		Bool;
OP120_Bypass_9:		Bool;
OP120_Bypass_10:    BOOL;
OP120_Bypass_11:    Bool;
OP120_Bypass_12:    Bool;
OP120_Bypass_13:    Bool;
OP120_Bypass_14:    Bool;
OP120_AnyBypass:	INT;

END_STRUCT
END_TYPE

// ---- POUs/Programs/OP120/OP120_Recipe.TcDUT
TYPE OP120_Recipe :
STRUCT
	OP120_Bowl_Feeder_Freq:LREAL;
	OP120_Robo_Prog_No:INT;
	OP120_Camera_Prog_No:INT;
	
END_STRUCT
END_TYPE

// ---- DUTs/OP10/OP10_GRP_CONTRL.TcDUT
TYPE OP10_GRP_CONTRL :
STRUCT
	LH_BODY_GRIP_WRK				: BOOL;
	LH_BODY_GRIP_HOM				: BOOL;	
	RH_BODY_GRIP_WRK				: BOOL;
	RH_BODY_GRIP_HME				: BOOL;
	LH_BODY_ROTRY_WRK				: BOOL;
	LH_BODY_RTRY_FITEE				: BOOL;	
	LH_BODY_ROTRY_CMR				: BOOL;	
	LH_BODY_ROTRY_HOM				: BOOL;	
	RH_BODY_ROTRY_WRK				: BOOL;
	RH_BODY_RTRY_FITEE				: BOOL;	
	RH_BODY_ROTRY_CMR				: BOOL;
	RH_BODY_ROTRY_HME				: BOOL;
	LH_BODY_GRIP_HOMING_1			: BOOL;
	RH_BODY_GRIP_HOMING_1			: BOOL;
	LH_BODY_ROTRY_HOMING_1			: BOOL;		
	RH_BODY_ROTRY_HOMING_1			: BOOL;	
END_STRUCT
END_TYPE

// ---- DUTs/OP10/OP10_GRP_STATUS.TcDUT
TYPE OP10_GRP_STATUS :
STRUCT
	LH_BDY_GRP_WRK_FB				: BOOL;
	LH_BDY_GRP_HOM_FB				: BOOL;	
	RH_BDY_GRP_WRK_FB				: BOOL;
	RH_BDY_GRP_HME_FB				: BOOL;
	LH_BDY_ROTRY_WRK_FB				: BOOL;
	LH_BDY_RTRY_FITEE_FB			: BOOL;	
	LH_BDY_ROTRY_CMR_FB				: BOOL;		
	LH_BDY_ROTRY_HOM_FB				: BOOL;	
	RH_BDY_ROTRY_WRK_FB				: BOOL;
	RH_BDY_RTRY_FITEE_FB			: BOOL;	
	RH_BDY_ROTRY_CMR_FB				: BOOL;			
	RH_BDY_ROTRY_HME_FB				: BOOL;
	LH_BDY_ROTRY_ZERO_FB			: BOOL;
	RH_BDY_ROTRY_ZERO_FB			: BOOL;
END_STRUCT
END_TYPE

// ---- DUTs/OP10/OP10_ORNG_CYL_DLY.TcDUT
TYPE OP10_ORNG_CYL_DLY :
STRUCT
	AFT_HORZ_FRW_DELY	: TIME;
	AFT_VERT_DWN_DELY	: TIME;
	AFT_GRP_WRK_DELY	: TIME;
	AFT_GRP_HME_DLY		: TIME;
	AFT_PSH_FRWD_DLY	: TIME;
	AFT_PSH_REV_DLY		: TIME;
	AFT_DEG_HME_DLY		: TIME;
	AFT_DEG_WRK_DLY		: TIME;	
END_STRUCT
END_TYPE

// ---- DUTs/OP10/OP10_ORNG_CYL_IP.TcDUT
TYPE OP10_ORNG_CYL_IP :
STRUCT
	HORIZ_CYL_SNR1			: BOOL;
	HORIZ_CYL_SNR2			: BOOL;	
	VERT_CYL_SNR1			: BOOL;
	VERT_CYL_SNR2			: BOOL;
	LH_O_GRP_SNR1			: BOOL;
	LH_O_GRP_SNR2			: BOOL;
	RH_O_GRP_SNR1			: BOOL;
	RH_O_GRP_SNR2			: BOOL;
	LH_O_PUSH_SNR1			: BOOL;
	LH_O_PUSH_SNR2			: BOOL;
	RH_O_PUSH_SNR1			: BOOL;
	RH_O_PUSH_SNR2			: BOOL;
	DEGREE_0				: BOOL;
	DEGREE_180				: BOOL;
	LH_REJ_SNR1				: BOOL;
	LH_REJ_SNR2				: BOOL;	
	RH_REJ_SNR1				: BOOL;
	RH_REJ_SNR2				: BOOL;		
END_STRUCT
END_TYPE

// ---- DUTs/OP10/OP10_ORNG_CYL_OP.TcDUT
TYPE OP10_ORNG_CYL_OP :
STRUCT
	HORIZ_CYL_AUT_CMD1			: BOOL;
	HORIZ_CYL_AUT_CMD2			: BOOL;	
	VERT_CYL_AUT_CMD1			: BOOL;
	VERT_CYL_AUT_CMD2			: BOOL;	
	LH_O_GRP_VALVE_ON			: BOOL;
	RH_O_GRP_VALVE_ON			: BOOL;
	LH_O_PSH_VALVE_ON			: BOOL;
	RH_O_PSH_VALVE_ON			: BOOL;
	DEGREE_AUT_CMD1				: BOOL;
	DEGREE_AUT_CMD2				: BOOL;	
	ALL_HOME					: BOOL;	
END_STRUCT
END_TYPE

// ---- DUTs/OP10/OP10_ROBO_CNTRL.TcDUT
TYPE OP10_ROBO_CNTRL :
STRUCT
	BDY_PCK_POSITION		: BOOL;
	BDY_S_PCK_POSITION		: BOOL;
	BDY_CMR_CHK_POS			: BOOL;
	BDY_S_ORNG_POS			: BOOL;
	BDY_ORNG_PLC_POS		: BOOL;
	BDY_MVE_PLC_POS			: BOOL;
	ROBO_SAFE_POS			: BOOL;
	ROBO_REJ_POS			: BOOL;
END_STRUCT
END_TYPE

// ---- DUTs/OP10/OP10_ROBO_STUS.TcDUT
TYPE OP10_ROBO_STUS :
STRUCT
	BDY_PCK_POSITION			: BOOL;
	BDY_S_PCK_POSITION			: BOOL;
	BDY_CMR_CHK_POS				: BOOL;
	BDY_S_ORNG_POS				: BOOL;
	BDY_ORNG_PLC_POS			: BOOL;
	BDY_MVE_PLC_POS				: BOOL;
	ROBO_SAFE_POS				: BOOL;
	ROBO_REJ_POS				: BOOL;
END_STRUCT
END_TYPE

// ---- DUTs/XTS/STATION_DONE.TcDUT
TYPE STATION_DONE :
STRUCT
		POSITION_DONE				: ARRAY[0..35] OF BOOL;
END_STRUCT
END_TYPE

// ---- FB/Axis/ENUM_Axis.TcDUT
{attribute 'qualified_only'}
{attribute 'strict'}
{attribute 'to_string'}
TYPE ENUM_Axis :

(
	Init := 0,
	PowerOFF,//Power off
	Error,
	Reset,
	PowerON,
	Stop,
	Halt,
	Ready,//Wait for command
	Homing,
	SetPosition,
	JogPos,
	JogNeg,
	MoveAbsolute,
	MoveRelative,
	MoveVelocity,
	MoveTorque
);	
	
END_TYPE

// ---- FB/Axis/OP10_SERVO_LIMIT.TcDUT
TYPE OP10_SERVO_LIMIT :
STRUCT	
OP10_FIRST_BODY_PIC_POS_LIMIT				: LREAL;
OP10_FIRST_BODY_PIC_NEG_LIMIT				: LREAL;
OP10_SECOND_BODY_PIC_POS_LIMIT				: LREAL;
OP10_SECOND_BODY_PIC_NEG_LIMIT				: LREAL;
OP10A_LH_GRPR_POS_LIMIT						: LREAL;
OP10A_LH_GRPR_NEG_LIMIT						: LREAL;
OP10A_LH_ROTRY_POS_LIMIT					: LREAL;
OP10A_LH_ROTRY_NEG_LIMIT					: LREAL;
OP10A_RH_GRPR_POS_LIMIT						: LREAL;
OP10A_RH_GRPR_NEG_LIMIT						: LREAL;
OP10A_RH_ROTRY_POS_LIMIT					: LREAL;
OP10A_RH_ROTRY_NEG_LIMIT					: LREAL;
OP10B_LH_GRPR_POS_LIMIT						: LREAL;
OP10B_LH_GRPR_NEG_LIMIT						: LREAL;
OP10B_LH_ROTRY_POS_LIMIT					: LREAL;
OP10B_LH_ROTRY_NEG_LIMIT					: LREAL;
OP10B_RH_GRPR_POS_LIMIT						: LREAL;
OP10B_RH_GRPR_NEG_LIMIT						: LREAL;
OP10B_RH_ROTRY_POS_LIMIT					: LREAL;
OP10B_RH_ROTRY_NEG_LIMIT					: LREAL;
OP10_FIRST_BODY_VELOCITY					: LREAL;
OP10_SECOND_BODY_VELOCITY					: LREAL;
OP10A_LH_GRPR_VELOCITY						: LREAL;
OP10A_LH_ROTRY_VELOCITY						: LREAL;
OP10A_RH_GRPR_VELOCITY						: LREAL;
OP10A_RH_ROTRY_VELOCITY						: LREAL;
OP10B_LH_GRPR_VELOCITY						: LREAL;
OP10B_LH_ROTRY_VELOCITY						: LREAL;
OP10B_RH_GRPR_VELOCITY						: LREAL;
OP10B_RH_ROTRY_VELOCITY						: LREAL;
END_STRUCT
END_TYPE

// ---- FB/Axis/OP90_SERVO_LIMIT.TcDUT
TYPE OP90_SERVO_LIMIT :
STRUCT
OP90_HORZ_POS_LIMIT					: LREAL;
OP90_HORZ_NEG_LIMIT                 : LREAL;
OP90_LH_VERT_POS_LIMIT              : LREAL;
OP90_LH_VERT_NEG_LIMIT              : LREAL;
OP90_RH_VERT_POS_LIMIT              : LREAL;
OP90_RH_VERT_NEG_LIMIT              : LREAL;
OP90_GUIDE_POS_LIMIT                : LREAL;
OP90_GUIDE_NEG_LIMIT                : LREAL;
OP90_LH_ROTRY_POS_LIMIT				: LREAL;
OP90_LH_ROTRY_NEG_LIMIT             : LREAL;
OP90_RH_ROTRY_POS_LIMIT				: LREAL;
OP90_RH_ROTRY_NEG_LIMIT             : LREAL;
OP90_A_HORZ_VELOCITY				: LREAL;
OP90_A_LH_VERT_VELOCITY             : LREAL;
OP90_A_RH_VERT_VELOCITY             : LREAL;
OP90_A_GUIDE_VELOCITY               : LREAL;
OP90_A_LH_ROTRY_VELOCITY			: LREAL;
OP90_A_RH_ROTRY_VELOCITY			: LREAL;
END_STRUCT
END_TYPE

// ---- FB/Axis/Servo_Control.TcDUT
TYPE Servo_Control :
STRUCT
	//input
	Reference_Start:BOOL;
	Reference_Position:LREAL;
	ABSmove_Start:BOOL;
	RELmove_Start:BOOL;
	VELmove_Start:BOOL;
	Torque_mode_Start:BOOL;
	Velocity: LREAL;	
	Position : LREAL; //target position
	BsetPos:BOOL;
	Bsethome : BOOL;
	Axis_Home_Cmd:BOOL;	
	Safety_cond : BOOL; //interlocks
	Axis_Home_Done : BOOL;
	//Output
	Axis_State:STRING;
	Axis_ready:BOOL;
	Axis_In_Pos:BOOL;
	Axis_Error:BOOL;
	Axis_Enabled:BOOL;
	Axis_reference:BOOL;
	Axis_In_Home: BOOL;
	Axis_Stopped:BOOL;
	Axis_Halted:BOOL;
	Safe_To_Move:BOOL;
	pos_done : BOOL;
	Trq_reached : BOOL;
	Actual_Position : LREAL;
	Actual_Velocity : LREAL;
	Actual_Torque : LREAL;
	
END_STRUCT
END_TYPE

// ---- FB/Axis/stManualModeAxis.TcDUT
TYPE stManualModeAxis :
STRUCT

stationModeAutoManual	: BOOL;
homing					: BOOL;
reset					: BOOL;
jogNeg					: BOOL;
jogPos					: BOOL;
moveAbsolute			: BOOL;
moveRelative			: BOOL;
moveVelocity			: BOOL;
moveTorque				: BOOL;
openBrake				: BOOL;
axisState				: STRING;
actualPosition			: LREAL;
actualVelocity			: LREAL;
targetPositon			: REAL;
targetVelocity			: REAL;



END_STRUCT
END_TYPE

// ---- FB/Cognex_Camera/Acquisition_control.TcDUT
TYPE Acquisition_control :
STRUCT
Trigger_Enable			: BIT;
Trigger					: BIT;
Clear_Exposure_Complete	: BIT;
Reserved3				: BIT;
Reserved4				: BIT;
Reserved5				: BIT;
Reserved6				: BIT;
Set_Offline				: BIT;
END_STRUCT
END_TYPE

// ---- FB/Cognex_Camera/Acquisition_status.TcDUT
TYPE Acquisition_status :
STRUCT
Trigger_Ready		: BIT ;
Trigger_Ack			: BIT ;
Exposure_Complete	: BIT ;
Missed_Ack			: BIT ;
Offline_Bit0		: BIT ;
Offline_Bit1		: BIT ;
Offline_Bit2		: BIT ;
Online				: BIT ;
END_STRUCT
END_TYPE

// ---- FB/Cognex_Camera/Inspection_control.TcDUT
TYPE Inspection_control :
STRUCT
Buffer_Results_Enable	: BIT ;
Inspection_Results_Ack	: BIT ;
Set_User_Data			: BIT ;
Execute_Command			: BIT ;
Reserved4				: BIT ;
Reserved5				: BIT ;
Reserved6				: BIT ;
Clear_Error				: BIT ;
END_STRUCT
END_TYPE

// ---- FB/Cognex_Camera/Inspection_status.TcDUT
TYPE Inspection_status :
STRUCT
System_Busy				: BIT ;
Inspection_Completed	: BIT ;
Results_Buffer_Overrun	: BIT ;
Results_Valid			: BIT ;
Command_Executing		: BIT ;
Command_Complete		: BIT ;
Command_Failed			: BIT ;
Set_User_Data_Ack		: BIT ;
Job_Pass				: BIT ;
Test_Run_Ready			: BIT ;
Reserved2				: BIT ;
Reserved3				: BIT ;
Reserved4				: BIT ;
Reserved5				: BIT ;
Reserved6				: BIT ;
Error					: BIT ;
END_STRUCT
END_TYPE

// ---- FB/Cognex_Camera/UNION_64Byte.TcDUT
TYPE UNION_64Byte :
UNION
sString 		: STRING(63);
aArrayOfByte 	: ARRAY[0..63] OF BYTE;
END_UNION
END_TYPE

// ---- FB/RFID/Head1.TcDUT
TYPE Head1 :
STRUCT
TimeoutActive:				BOOL;
NewData:					BOOL;
NotExist:					BOOL;
ExistTC:					BOOL;
Error:						BOOL;
TimeoutOccurred:			BOOL;
SendOK:						BOOL;
ReceiveOK:					BOOL;
NoDataCarrier:				BOOL;
Busy:						BOOL;
Done:						BOOL;
EnhCommandActive:			BOOL;
SglCommandActive:			BOOL;
TransfToHead:				BOOL;
Execute:					BOOL;
SaveRead:					BOOL;
SaveWrite:					BOOL;
SaveQuit:					BOOL;
SaveSpecialCommand:			BOOL;
END_STRUCT
END_TYPE

// ---- FB/RFID/HeadData.TcDUT
TYPE HeadData :
STRUCT
WriteData:	 	ARRAY [0..63] OF BYTE;	
ReadData:		ARRAY [0..63] OF BYTE;
SpecialCommand:	ARRAY [0..63] OF BYTE;
END_STRUCT
END_TYPE

// ---- FB/RFID/Memory.TcDUT
TYPE Memory :
STRUCT

Memory:				ARRAY [0..63] OF BYTE;	
OldCommandIn:		BYTE;
OldChannelIn:		BYTE;
OldStatus:			BYTE;
OldReplyCounter:	BYTE;
Headnumber:			USINT;
Togglebit:			USINT;


END_STRUCT
END_TYPE

// ---- FB/RFID/UNION_RFID.TcDUT
TYPE UNION_RFID :
UNION
	aArray		: ARRAY[0..63] OF BYTE;
	Number		: UDINT;
END_UNION
END_TYPE

// ---- FB/Robot/E_State_RobotGeneral.TcDUT
{attribute 'qualified_only'}
{attribute 'strict'}
{attribute 'to_string'}
TYPE E_State_RobotGeneral :
(
	Init := 0,
	AutoEnable,
	OperationEnable,
	Error,
	ErrorReset,
	ServoOn,
	Start,
	Started,
	ProgramStop,
	ProgramReset
	
);
END_TYPE

// ---- FB/Scanner/Acquisition_Control_Scanner.TcDUT
TYPE Acquisition_Control_Scanner :
STRUCT
	Trigger_Enable : BOOL;
	Trigger		   : BOOL;
END_STRUCT
END_TYPE

// ---- FB/Scanner/Acquisition_Status_Scanner.TcDUT
TYPE Acquisition_Status_Scanner  :
STRUCT
	Trigger_ready		: BOOL;
	Triger_Acknowledge  : BOOL;
	Acquiring 			: BOOL;
END_STRUCT
END_TYPE

// ---- FB/Scanner/Result_Control_Scanner.TcDUT
TYPE Result_Control_Scanner :
STRUCT
	Enable_Result_Buffering : BOOL;
	Result_Acknowledge		: BOOL;
END_STRUCT
END_TYPE

// ---- FB/Scanner/Result_Data_Register.TcDUT
TYPE Result_Data_Register :
STRUCT
	Result_ID 		: UINT;
	Result_Code		: UINT;
	Result_Extended : UINT;
	Result_Length   : UINT;
END_STRUCT
END_TYPE

// ---- FB/Scanner/Result_Status.TcDUT
TYPE Result_Status :
STRUCT
	Decoding			  : BOOL;
	Decode_Complete 	  : BOOL;
	Result_Buffer_overrun : BOOL;
	Result_Available	  : BOOL;
	Set_When_fault_Occur  : BOOL;
END_STRUCT
END_TYPE

// ---- FB/Schunk/ENUM_Schunk.TcDUT
{attribute 'qualified_only'}
{attribute 'strict'}
{attribute 'to_string'}
TYPE ENUM_Schunk :

(
	Init := 0,
	Undefined,
	Error,
	Reset,
	Stop,
	Ready,//Wait for command
	Homing,
	SetPosition,
	MoveAbsolute,
	MoveRelative
);	
	
END_TYPE

// ---- FB/Schunk/iSchunkProcessData.TcDUT
TYPE iSchunkProcessData :
STRUCT
	
commandReleaseA:			BIT;
commandReleaseB:			BIT;
spare1:						BIT;
spare2:						BIT;
spare3:						BIT;
spare4:						BIT;
moduleReady:				BIT;
spare5:						BIT;
moduleIsMoving:				BIT;
targetPosReached:			BIT;
movementBlocked:			BIT;
brakeActive:				BIT;
modulIsReferenced:			BIT;
info:						BIT;
warning:					BIT;
error:						BIT;
activeCopy:					BYTE;
digitalInputs:				BYTE;
actualPos:					REAL;
actualVelo:					REAL;
actualCurrent:				REAL;
errorCode:					BYTE;
notUsed:					BYTE;


END_STRUCT
END_TYPE

// ---- FB/Schunk/oSchunkProcessData.TcDUT
TYPE oSchunkProcessData :
STRUCT

commandReleaseA:				BIT;
commandReleaseB:				BIT;
jerkActivate:					BIT;
currentActivate:				BIT;
accelerationActivate:			BIT;
velocityMove:					BIT;
moveToPosition:					BIT;
moveToRelativePosition:			BIT;
spare1:							BIT;
modulReference:					BIT;
spare2:							BIT;
spare3:							BIT;
restartModul:					BIT;
ackError:						BIT;
stop:							BIT;
fastStop:						BIT;
notUsed:						BYTE;
digitalOutputs:					BYTE;
targetPos:						REAL;
targetVelo:						REAL;
targetCurrent:					REAL;
targetAcc:						REAL;
targetJerk:						REAL;
	
END_STRUCT
END_TYPE

// ---- FB/Schunk/stManualModeAxis_1.TcDUT
TYPE stManualModeAxis_1 :
STRUCT

stationModeAutoManual	: BOOL;
homing					: BOOL;
reset					: BOOL;
jogNeg					: BOOL;
jogPos					: BOOL;
moveAbsolute			: BOOL;
moveRelative			: BOOL;
moveVelocity			: BOOL;
openBrake				: BOOL;
axisState				: STRING;
actualPosition			: LREAL;
actualVelocity			: LREAL;
targetPositon			: REAL;
targetVelocity			: REAL;



END_STRUCT
END_TYPE

// ---- FB/Schunk/UNION_iSchunkProcessData.TcDUT
TYPE UNION_iSchunkProcessData :
UNION
	Schunk_in 		: ARRAY [0..8] OF WORD;
	iSchunk_ProcessData	: iSchunkProcessData;
END_UNION
END_TYPE

// ---- FB/Schunk/UNION_oSchunkProcessData.TcDUT
TYPE UNION_oSchunkProcessData :
UNION
	Schunk_out 		: ARRAY [0..11] OF WORD;
	oSchunk_ProcessData	: oSchunkProcessData;
END_UNION
END_TYPE

// ---- FB/Schunk/UNION_REAL.TcDUT
TYPE UNION_REAL :
UNION
	rREAL	: REAL;
	aARRAY	: ARRAY[0..3]OF BYTE;
END_UNION
END_TYPE

// ---- GVLs/E_EcCommState.TcDUT
TYPE E_EcCommState : (
	UNDEFINED 	:= 0,
	INIT 			:= 1,
	PREOP 		:= 2,
	BOOT 			:= 3,
	SAFEOP 		:= 4,
	OP 			:= 8
);
END_TYPE

// ---- GVLs/ST_SlaveState.TcDUT
TYPE ST_SlaveState :
STRUCT
		(* slave state *)
	eEcState 		: E_EcCommState;
	nReserved		: UINT;
	bError			: BOOL;
	bInvalidVPRS	: BOOL;
	nReserved2		: UINT;

	(* link state *)
	bNoCommToSlave	: BOOL;
	bLinkError		: BOOL;
	bMissingLink	: BOOL;
	bUnexpectedLink	: BOOL;
	bPortA			: BOOL;
	bPortB			: BOOL;
	bPortC			: BOOL;
	bPortD			: BOOL;
END_STRUCT
END_TYPE

// ---- POUs/Programs/OP130/OP130_Recipe.TcDUT
TYPE OP130_Recipe :
STRUCT


END_STRUCT
END_TYPE

// ---- POUs/Programs/OP160/OP160_Recipe.TcDUT
TYPE OP160_Recipe :
STRUCT
	OP160_Robo_Prog_No:INT;
END_STRUCT
END_TYPE

// ---- POUs/Programs/OP10/OP10_HMI_GVL.TcGVL
//{attribute 'qualified_only'}
VAR_GLOBAL

	
//LREAL
	OP10A_SRV_ACT_POS								: LREAL;
	OP10B_SRV_ACT_POS								: LREAL;
//REAL
	OP10A_TARGET_POSITION							: REAL;
	OP10A_TARGET_VEL								: REAL;
	OP10B_TARGET_POSITION							: REAL;
//INT 
	OP10_CYL_NO										: INT;
	OP10B_CYL_NO									: INT;	
	OP10_SERVO_NO									: INT;
	OP10B_SERVO_NO									: INT;
	OP10A_AUTO_STATUS_MES							: INT;	
	OP10B_AUTO_STATUS_MES							: INT;	
//BOOL
	OP10_HOME										: BOOL;
	OP10_WORK										: BOOL;
	OP10B_HOME										: BOOL;
	OP10B_WORK										: BOOL;	
	OP10_JOG_POSITIVE								: BOOL;
	OP10_JOG_NEGATIVE								: BOOL;
	OP10B_JOG_POSITIVE								: BOOL;
	OP10B_JOG_NEGATIVE								: BOOL;
	OP10A_SET_HOME									: BOOL;
	OP10B_SET_HOME									: BOOL;
	OP10A_MOVE_TARGET								: BOOL;
	OP10A_SRV_FAULT									: BOOL;	
	OP10B_SRV_FAULT									: BOOL;
	OP10B_SRV_ENABLE								: BOOL;
	OP10B_MOVE_TARGET								: BOOL;
	OP10A_SRV_ENABLE								: BOOL;
	OP10A_STRT_PB									: BOOL;
	OP10B_STRT_PB									: BOOL;	
// ROBO
									(*OP10A*)
	OP10A_M_BODY_READY_TO_PICK						: BOOL;
	OP10A_M_PICK_PART_OK							: BOOL;
	OP10A_M_PICK_PART_NOK                           : BOOL;
	OP10A_M_CAMERA_OK                               : BOOL;
	OP10A_M_CAMERA_NOK                              : BOOL;
	OP10A_M_GRIPPER_ROTATE_COMPLETE                 : BOOL;
	OP10A_M_READY_TO_INSERT_ORING                   : BOOL;
	OP10A_M_ORING_INSERTION_DONE                    : BOOL;
	OP10A_M_PLACE_IN_CONVEYOR                       : BOOL;
	OP10A_M_PLACE_IN_REJECTION                      : BOOL;
	OP10A_M_GRIPPER_OPEN                            : BOOL;
	OP10A_M_GRIPPER_CLOSE                           : BOOL;
									(*OP10B*)	
	OP10B_M_BODY_READY_TO_PICK						: BOOL;
	OP10B_M_PICK_PART_OK							: BOOL;
	OP10B_M_PICK_PART_NOK                           : BOOL;
	OP10B_M_CAMERA_OK                               : BOOL;
	OP10B_M_CAMERA_NOK                              : BOOL;
	OP10B_M_GRIPPER_ROTATE_COMPLETE                 : BOOL;
	OP10B_M_READY_TO_INSERT_ORING                   : BOOL;
	OP10B_M_ORING_INSERTION_DONE                    : BOOL;
	OP10B_M_PLACE_IN_CONVEYOR                       : BOOL;
	OP10B_M_PLACE_IN_REJECTION                      : BOOL;
	OP10B_M_GRIPPER_OPEN                            : BOOL;
	OP10B_M_GRIPPER_CLOSE                           : BOOL;	
	


	
END_VAR





VAR_GLOBAL PERSISTENT
	OP10_SERVO_POS_VEL_LIMIT: OP10_SERVO_LIMIT;
END_VAR

// ---- POUs/Programs/OP10/OP10_VARIABLE.TcGVL
VAR_GLOBAL
// FUNCTIONAL BLOCK
									(*CYLINDER*)
	OP10A_HORZ_CYL									: Cylinder_Block_HOMING;
	OP10A_VERT_CYL									: Cylinder_Block_HOMING;	
	OP10A_DEGREE_CYL								: Cylinder_Block_HOMING;
	OP10A_LH_GRP									: Cylinder_Block_HOMING;
	OP10A_RH_GRP                                    : Cylinder_Block_HOMING;
	OP10A_LH_PUSH                                   : Cylinder_Block_HOMING;
	OP10A_RH_PUSH									: Cylinder_Block_HOMING;
	OP10B_HORZ_CYL									: Cylinder_Block_HOMING;
	OP10B_VERT_CYL									: Cylinder_Block_HOMING;	
	OP10B_DEGREE_CYL								: Cylinder_Block_HOMING;
	OP10B_LH_GRP									: Cylinder_Block_HOMING;
	OP10B_RH_GRP                                    : Cylinder_Block_HOMING;
	OP10B_LH_PUSH                                   : Cylinder_Block_HOMING;
	OP10B_RH_PUSH									: Cylinder_Block_HOMING;
	OP10B_LH_REJ                                    : Cylinder_Block_HOMING;
	OP10B_RH_REJ									: Cylinder_Block_HOMING;	
	OP10A_LH_REJ                                    : Cylinder_Block_HOMING;
	OP10A_RH_REJ									: Cylinder_Block_HOMING;
	OP10_BDY_SING_FRT                               : Cylinder_Block_HOMING;
	OP10_BDY_SING_SEC								: Cylinder_Block_HOMING;


// ROBO
									(*OP10A*)
	OP10A_ROBO_MODE_NO AT %Q*						: UINT;
	OP10A_ROBO_VARIENT AT %Q*						: UINT	:=1;
	OP10A_ROBO_STATUS								: OP10_ROBO_STUS;
	OP10A_ROBO_CNTRL								: OP10_ROBO_CNTRL;
	OP10A_GRP_STATUS								: OP10_GRP_STATUS;
	OP10A_GRP_CNTRL									: OP10_GRP_CONTRL;								
	OP10A_ROBO_PRGM_RST								: BOOL;
    OP10A_A_BODY_READY_TO_PICK						: BOOL;
    OP10A_A_PICK_PART_OK							: BOOL;
    OP10A_A_PICK_PART_NOK                           : BOOL;
    OP10A_A_CAMERA_OK                               : BOOL;
    OP10A_A_CAMERA_NOK                              : BOOL;
    OP10A_A_GRIPPER_ROTATE_COMPLETE                 : BOOL;
    OP10A_A_READY_TO_INSERT_ORING                   : BOOL;
    OP10A_A_ORING_INSERTION_DONE                    : BOOL;
    OP10A_A_PLACE_IN_CONVEYOR                       : BOOL;
    OP10A_A_PLACE_IN_REJECTION                      : BOOL;
    OP10A_A_GRIPPER_OPEN                            : BOOL;
    OP10A_A_GRIPPER_CLOSE                           : BOOL;
    OP10A_BODY_READY_TO_PICK						: BOOL;
    OP10A_PICK_PART_OK								: BOOL;
    OP10A_PICK_PART_NOK                           	: BOOL;
    OP10A_CAMERA_OK                               	: BOOL;
    OP10A_CAMERA_NOK                              	: BOOL;
    OP10A_GRIPPER_ROTATE_COMPLETE                 	: BOOL;
    OP10A_READY_TO_INSERT_ORING                   	: BOOL;
    OP10A_ORING_INSERTION_DONE                    	: BOOL;
    OP10A_PLACE_IN_CONVEYOR                       	: BOOL;
    OP10A_PLACE_IN_REJECTION                      	: BOOL;
	OP10A_ROTATION_COMPLETE							: BOOL;
	WITH_ORING_VARIIENT								: BOOL;
    OP10A_GRIPPER_OPEN                            	: BOOL;
    OP10A_GRIPPER_CLOSE                           	: BOOL;
	OP10A_AUTO_ENABLE								: BOOL;
	OP10A_START										: BOOL;
	OP10A_STOP										: BOOL;
	OP10A_STOP2										: BOOL;
	OP10A_PRGM_RST									: BOOL;
	OP10A_ERR_RST									: BOOL;
	OP10A_CYCLE_STP									: BOOL;
	OP10A_SERVO_OFF									: BOOL;
	OP10A_SERVO_ON									: BOOL;
	OP10A_OPERATION_ENABLE							: BOOL;
	OP10A_MOVER_HOME								: BOOL;
	OP10A_General_Output_reset						: BOOL;
	OP10A_Machine_Lock								: BOOL;
	OP10A_PLC_Heartbeat								: BOOL;
	OP10A_Homing_Start								: BOOL;
	OP10A_Pick_Zone_Safe							: BOOL;
	OP10A_Camera_Zone_Safe							: BOOL;
	OP10A_O_Ring_Zone_Safe							: BOOL;
	OP10A_Place_Zone_Safe							: BOOL;
	OP10A_Reject_Zone_Safe							: BOOL;
	OP10A_Robot2_In_Pick_Sequence					: BOOL;
	OP10_A_FRT_BDY_SING_WRK							: BOOL;
	OP10_A_SEC_BDY_SING_WRK							: BOOL;
	OP10_A_FRT_BDY_SING_HME							: BOOL;
	OP10_A_SEC_BDY_SING_HME							: BOOL;
	OP10A_Mirror_Auto_enable						: BOOL;
	OP10A_Program_Execute							: BOOL;
	OP10A_Program_Waiting							: BOOL;
	OP10A_Program_Waiting2							: BOOL;
	OP10A_Stop_Status								: BOOL;
	OP10A_Program_Sel_enabled_OP					: BOOL;
	OP10A_During_error								: BOOL;
	OP10A_During_Cycle_Stop							: BOOL;
	OP10A_Mirror_SRVO_Off							: BOOL;
	OP10A_Servo_ON_OFF_Status						: BOOL;
	OP10A_Auto_Operation_Enable						: BOOL;
	OP10A_Moving_Home								: BOOL;
	OP10A_Spare1									: BOOL;
	OP10A_During_Machine_Lock						: BOOL;
	OP10A_H_Error									: BOOL;
	OP10A_L_Error									: BOOL;
	OP10A_Caution									: BOOL;
	OP10A_During_EMG_Stop							: BOOL;
	OP10A_Teach_Mode								: BOOL;
	OP10A_Auto_OP_Mode								: BOOL;
	OP10A_Auto_Ext_Mode								: BOOL;
	OP10A_TP_Enable									: BOOL;
	OP10A_Heartbeat									: BOOL;
	OP10A_Spare2									: BOOL;
	OP10A_Rbt_In_Home								: BOOL;
	OP10A_Rbt_In_Pick_Zone							: BOOL;
	OP10A_Rbt_In_Camera_Zone						: BOOL;
	OP10A_Rbt_In_O_Ring_Zone						: BOOL;
	OP10A_Rbt_In_Place_Zone							: BOOL;
	OP10A_Rbt_In_Reject_Zone						: BOOL;
	OP10A_Spare7									: BOOL;
	OP10A_Robot1_In_Pick_Sequence					: BOOL;
	OP10A_Sequence_Running							: BOOL;
	OP10A_Sequence_Completed						: BOOL;
	OP10A_Part_Pick_Completed						: BOOL;
	OP10A_Spare10									: BOOL;
	OP10A_NOK_Part_Dropped							: BOOL;
	OP10A_Spare11									: BOOL;
	OP10A_Camera_Trigger							: BOOL;
	OP10A_Spare12									: BOOL;
	OP10A_O_Ring_Pick_Pos_Reached					: BOOL;
	OP10A_Spare13									: BOOL;
	OP10A_Part_Place_Conveyor						: BOOL;
	OP10A_Spare5									: BOOL;
	OP10A_Spare6									: BOOL;
	OP10A_Step_Reached								: BOOL;
	OP10A_StartOf_Sequence							: BOOL;
	OP10A_ROBO_Gripper_Open							: BOOL;
	OP10A_ROBO_Gripper_Close						: BOOL;
	OP10A_Spare14									: BOOL;
	OP10A_Spare15									: BOOL;
	OP10A_Spare16									: BOOL;
	OP10A_Spare17									: BOOL;
	OP10A_Spare18									: BOOL;
	OP10A_Spare19									: BOOL;
	OP10A_Spare27									: BOOL;
	OP10A_Spare26									: BOOL;
	OP10A_CMP_PRS_ROBO								: BOOL;
	OP10A_Spare24									: BOOL;
	OP10A_Spare23									: BOOL;
	OP10A_Spare22									: BOOL;
	OP10A_Spare21									: BOOL;
	OP10A_Spare20									: BOOL;

	
   								(*OP10B*)
	OP10B_ROBO_MODE_NO AT %Q*						: UINT;
	OP10B_ROBO_VARIENT AT %Q*						: UINT	:=1;
	OP10B_ROBO_STATUS								: OP10_ROBO_STUS;
	OP10B_GRP_STATUS								: OP10_GRP_STATUS;
	OP10B_GRP_CNTRL									: OP10_GRP_CONTRL;							
	OP10B_ROBO_CNTRL								: OP10_ROBO_CNTRL;
	OP10B_ROBO_PRGM_RST								: BOOL;	
    OP10B_A_BODY_READY_TO_PICK						: BOOL;
    OP10B_A_PICK_PART_OK							: BOOL;
    OP10B_A_PICK_PART_NOK                           : BOOL;
    OP10B_A_CAMERA_OK                               : BOOL;
    OP10B_A_CAMERA_NOK                              : BOOL;
    OP10B_A_GRIPPER_ROTATE_COMPLETE                 : BOOL;
    OP10B_A_READY_TO_INSERT_ORING                   : BOOL;
    OP10B_A_ORING_INSERTION_DONE                    : BOOL;
    OP10B_A_PLACE_IN_CONVEYOR                       : BOOL;
    OP10B_A_PLACE_IN_REJECTION                      : BOOL;
    OP10B_A_GRIPPER_OPEN                            : BOOL;
    OP10B_A_GRIPPER_CLOSE                           : BOOL;
	OP10B_ROTATION_COMPLETE							: BOOL;
    OP10B_BODY_READY_TO_PICK						: BOOL;
    OP10B_PICK_PART_OK								: BOOL;
    OP10B_PICK_PART_NOK                           	: BOOL;
    OP10B_CAMERA_OK                               	: BOOL;
    OP10B_CAMERA_NOK                              	: BOOL;
    OP10B_GRIPPER_ROTATE_COMPLETE                 	: BOOL;
    OP10B_READY_TO_INSERT_ORING                   	: BOOL;
    OP10B_ORING_INSERTION_DONE                    	: BOOL;
    OP10B_PLACE_IN_CONVEYOR                       	: BOOL;
    OP10B_PLACE_IN_REJECTION                      	: BOOL;
    OP10B_GRIPPER_OPEN                            	: BOOL;
    OP10B_GRIPPER_CLOSE                           	: BOOL;	
	OP10B_AUTO_ENABLE								: BOOL;
	OP10B_START										: BOOL;
	OP10B_STOP										: BOOL;
	OP10B_STOP2										: BOOL;
	OP10B_PRGM_RST									: BOOL;
	OP10B_ERR_RST									: BOOL;
	OP10B_CYCLE_STP									: BOOL;
	OP10B_SERVO_OFF									: BOOL;
	OP10B_SERVO_ON									: BOOL;
	OP10B_OPERATION_ENABLE							: BOOL;
	OP10B_MOVER_HOME								: BOOL;
	OP10B_General_Output_reset						: BOOL;
	OP10B_Machine_Lock								: BOOL;
	OP10B_PLC_Heartbeat								: BOOL;
	OP10B_Homing_Start								: BOOL;
	OP10B_Pick_Zone_Safe							: BOOL;
	OP10B_Camera_Zone_Safe							: BOOL;
	OP10B_O_Ring_Zone_Safe							: BOOL;
	OP10B_Place_Zone_Safe							: BOOL;
	OP10B_Reject_Zone_Safe							: BOOL;
	OP10B_Robot2_In_Pick_Sequence					: BOOL;	

	OP10B_Mirror_Auto_enable						: BOOL;
	OP10B_Program_Execute							: BOOL;
	OP10B_Program_Waiting							: BOOL;
	OP10B_Program_Waiting2							: BOOL;
	OP10B_Stop_Status								: BOOL;
	OP10B_Program_Sel_enabled_OP					: BOOL;
	OP10B_During_error								: BOOL;
	OP10B_During_Cycle_Stop							: BOOL;
	OP10B_Mirror_SRVO_Off							: BOOL;
	OP10B_Servo_ON_OFF_Status						: BOOL;
	OP10B_Auto_Operation_Enable						: BOOL;
	OP10B_Moving_Home								: BOOL;
	OP10B_Spare1									: BOOL;
	OP10B_During_Machine_Lock						: BOOL;
	OP10B_H_Error									: BOOL;
	OP10B_L_Error									: BOOL;
	OP10B_Caution									: BOOL;
	OP10B_During_EMG_Stop							: BOOL;
	OP10B_Teach_Mode								: BOOL;
	OP10B_Auto_OP_Mode								: BOOL;
	OP10B_Auto_Ext_Mode								: BOOL;
	OP10B_TP_Enable									: BOOL;
	OP10B_Heartbeat									: BOOL;
	OP10B_Spare2									: BOOL;
	OP10B_Rbt_In_Home								: BOOL;
	OP10B_Rbt_In_Pick_Zone							: BOOL;
	OP10B_Rbt_In_Camera_Zone						: BOOL;
	OP10B_Rbt_In_O_Ring_Zone						: BOOL;
	OP10B_Rbt_In_Place_Zone							: BOOL;
	OP10B_Rbt_In_Reject_Zone						: BOOL;
	OP10B_Spare7									: BOOL;
	OP10B_Robot1_In_Pick_Sequence					: BOOL;
	OP10B_Sequence_Running							: BOOL;
	OP10B_Sequence_Completed						: BOOL;
	OP10B_Part_Pick_Completed						: BOOL;
	OP10B_Spare10									: BOOL;
	OP10B_NOK_Part_Dropped							: BOOL;
	OP10B_Spare11									: BOOL;
	OP10B_Camera_Trigger							: BOOL;
	OP10B_Spare12									: BOOL;
	OP10B_O_Ring_Pick_Pos_Reached					: BOOL;
	OP10B_Spare13									: BOOL;
	OP10B_Part_Place_Conveyor						: BOOL;
	OP10B_Spare5									: BOOL;
	OP10B_Spare6									: BOOL;
	OP10B_Step_Reached								: BOOL;
	OP10B_StartOf_Sequence							: BOOL;
	OP10B_ROBO_Gripper_Open							: BOOL;
	OP10B_ROBO_Gripper_Close						: BOOL;
	OP10B_Spare14									: BOOL;
	OP10B_Spare15									: BOOL;
	OP10B_Spare16									: BOOL;
	OP10B_Spare17									: BOOL;
	OP10B_Spare18									: BOOL;
	OP10B_Spare19									: BOOL;
	OP10B_Spare27									: BOOL;
	OP10B_Spare26									: BOOL;
	OP10B_CMP_PRS_ROBO								: BOOL;
	OP10B_Spare24									: BOOL;
	OP10B_Spare23									: BOOL;
	OP10B_Spare22									: BOOL;
	OP10B_Spare21									: BOOL;
	OP10B_Spare20									: BOOL;	
	
									(*SERVO*)
									(*OP10*)
									
	OP10_SRV_FRST_PCKBDY_CNT						: Servo_Control;
	OP10_SRV_SCND_PCKBDY_CNT						: Servo_Control;
	OP10_SRV_FRST_PCKBDY_STUS						: stManualModeAxis;
	OP10_SRV_SCND_PCKBDY_STUS						: stManualModeAxis;
	OP10_FRT_BDY_GPR								: FB_Axis_FESTO;
	OP10_SEC_BDY_GPR								: FB_Axis_FESTO;
	OP10_A_SRV_FST_BDYPCK_WRK						: BOOL;
	OP10_A_SRV_FST_BDYPCK_HME						: BOOL;
	OP10_A_SRV_SCND_BDYPCK_WRK						: BOOL;
	OP10_A_SRV_SCND_BDYPCK_HME						: BOOL;	
/////////////////				(*SERVO_OP10A*)
	OP10A_LH_ROTY									: FB_Axis_FESTO;
	OP10A_RH_ROTY									: FB_Axis_FESTO;
	OP10A_LH_GRIPR									: FB_Axis_FESTO;
	OP10A_RH_GRIPR									: FB_Axis_FESTO;
	OP10A_CONVEYOR									: FB_Axis;	
	OP10A_SRV_LH_BDYANG_CNT							: SERVO_Control;
	OP10A_SRV_RH_BDYANG_CNT                     	: SERVO_Control;
	OP10A_SRV_LH_BDYGRP_CNT                     	: SERVO_Control;
	OP10A_SRV_RH_BDYGRP_CNT                     	: SERVO_Control;
	OP10A_SRV_O_CNVY_CNT                        	: SERVO_Control;
	OP10A_SRV_LH_BDYANG_STUS						: stManualModeAxis;	
	OP10A_SRV_RH_BDYANG_STUS                    	: stManualModeAxis;	
	OP10A_SRV_LH_BDYGRP_STUS                    	: stManualModeAxis;	
	OP10A_SRV_RH_BDYGRP_STUS                    	: stManualModeAxis;	
	OP10A_SRV_O_CNVY_STUS	                    	: stManualModeAxis;
	OP10A_A_SRV_LH_GRPWRK							: BOOL;
	OP10A_A_SRV_LH_GRPHME							: BOOL;
	OP10A_A_SRV_RH_GRPWRK							: BOOL;
	OP10A_A_SRV_RH_GRPHME							: BOOL;
	OP10A_SRV_LH_BDYANG_HME							: BOOL;	
	OP10A_SRV_LH_BDYANG_CMR							: BOOL;	
	OP10A_SRV_LH_BDYANG_FITRE						: BOOL;		
	OP10A_SRV_LH_BDYANG_WRK							: BOOL;
	OP10A_SRV_RH_BDYANG_HME							: BOOL;
	OP10A_SRV_RH_BDYANG_CMR							: BOOL;
	OP10A_SRV_RH_BDYANG_FITRE						: BOOL;	
	
	OP10A_SRV_RH_BDYANG_WRK							: BOOL;
	OP10B_A_SRV_LH_GRPWRK							: BOOL;
	OP10B_A_SRV_LH_GRPHME							: BOOL;
	OP10B_A_SRV_RH_GRPWRK							: BOOL;
	OP10B_A_SRV_RH_GRPHME							: BOOL;
	OP10B_SRV_LH_BDYANG_HME							: BOOL;
	OP10B_SRV_LH_BDYANG_CMR							: BOOL;
	OP10B_SRV_LH_BDYANG_FITRE						: BOOL;	
	OP10B_SRV_LH_BDYANG_WRK							: BOOL;
	OP10B_SRV_RH_BDYANG_HME							: BOOL;
	OP10B_SRV_RH_BDYANG_CMR							: BOOL;
	OP10B_SRV_RH_BDYANG_FITRE						: BOOL;	
	OP10B_SRV_RH_BDYANG_WRK							: BOOL;	
/////////////////				(*SERVO_OP10B*) 
	OP10B_LH_ROTY									: FB_Axis_FESTO;
	OP10B_RH_ROTY									: FB_Axis_FESTO;
	OP10B_LH_GRIPR									: FB_Axis_FESTO;
	OP10B_RH_GRIPR									: FB_Axis_FESTO;
	OP10B_CONVEYOR									: FB_Axis;	                            	
	OP10B_SRV_LH_BDYANG_CNT							: SERVO_Control;
	OP10B_SRV_RH_BDYANG_CNT                     	: SERVO_Control;
	OP10B_SRV_LH_BDYGRP_CNT                     	: SERVO_Control;
	OP10B_SRV_RH_BDYGRP_CNT                     	: SERVO_Control;
	OP10B_SRV_O_CNVY_CNT                            : SERVO_Control;
	OP10B_SRV_LH_BDYANG_STUS						: stManualModeAxis;	
	OP10B_SRV_RH_BDYANG_STUS                    	: stManualModeAxis;	
	OP10B_SRV_LH_BDYGRP_STUS                    	: stManualModeAxis;	
	OP10B_SRV_RH_BDYGRP_STUS                    	: stManualModeAxis;	
	OP10B_SRV_O_CNVY_STUS	                        : stManualModeAxis;
	OP10_SRV_FRST_PCKBDY_WRK_FB						: BOOL;
	OP10_SRV_FRST_PCKBDY_HME_FB						: BOOL;
	OP10_SRV_SCND_PCKBDY_WRK_FB						: BOOL;	
	OP10_SRV_SCND_PCKBDY_HME_FB						: BOOL;	
	OP10A_A_SRV_RH_GRPWRK_FB						: BOOL;	
	OP10A_A_SRV_LH_GRPWRK_FB						: BOOL;	
	OP10A_A_SRV_RH_GRPHME_FB						: BOOL;
	OP10A_A_SRV_LH_GRPHME_FB						: BOOL;	
	OP10A_SRV_LH_BDYANG_HME_FB						: BOOL;
	OP10A_SRV_RH_BDYANG_HME_FB						: BOOL;
	OP10A_SRV_RH_BDYANG_CMR_FB						: BOOL;
	OP10A_SRV_RH_BDYANG_FITRE_FB					: BOOL;
	OP10A_SRV_LH_BDYANG_CMR_FB						: BOOL;
	OP10A_SRV_LH_BDYANG_FITRE_FB					: BOOL;	

	
	OP10A_SRV_LH_BDYANG_WRK_FB						: BOOL;
	OP10A_SRV_RH_BDYANG_WRK_FB						: BOOL;
	OP10A_SRV_RH_BDYANG_ZERO_FB						: BOOL;
	OP10A_SRV_LH_BDYANG_ZERO_FB						: BOOL;
	OP10B_A_SRV_LH_GRPWRK_FB						: BOOL;
	OP10B_A_SRV_LH_GRPHME_FB						: BOOL;
	OP10B_A_SRV_RH_GRPWRK_FB						: BOOL;
	OP10B_A_SRV_RH_GRPHME_FB						: BOOL;
	OP10B_SRV_LH_BDYANG_HME_FB						: BOOL;
	OP10B_SRV_LH_BDYANG_CMR_FB						: BOOL;	
	OP10B_SRV_LH_BDYANG_FITRE_FB					: BOOL;
	OP10B_SRV_LH_BDYANG_WRK_FB						: BOOL;
	OP10B_SRV_RH_BDYANG_HME_FB						: BOOL;
	OP10B_SRV_RH_BDYANG_CMR_FB						: BOOL;
	OP10B_SRV_RH_BDYANG_FITRE_FB					: BOOL;
	OP10B_SRV_RH_BDYANG_WRK_FB						: BOOL;
	OP10B_SRV_RH_BDYANG_ZERO_FB						: BOOL;
	OP10B_SRV_LH_BDYANG_ZERO_FB						: BOOL;
		
// HOMING

	OP10_FRT_CYL_INITZAL							: BOOL;
	OP10_SEC_CYL_INITZAL							: BOOL;
									(*OP10A*)
	R1												: R_TRIG;							
	OP10A_START_HOMNG								: BOOL;
	OP10A_GRIPPER_HOME								: BOOL;	
	OP10A_O_LHGRIP_HMG1								: BOOL;
	OP10A_O_RHGRIP_HMG1								: BOOL;
	OP10A_O_LHPUSH_HMG1								: BOOL;
	OP10A_O_RHPUSH_HMG1								: BOOL;
	OP10A_O_VERT_HMG1								: BOOL;
	OP10A_O_DEGRE_HMG1								: BOOL;
	OP10A_O_HORZ_HMG1								: BOOL;
	OP10A_ALL_HOME									: BOOL;
	OP10A_ROBO_SFE_HME								: BOOL;	
	OP10A_ROBO_SFE_HME_FB							: BOOL;	
	OP10A_GRP_REFERENCED							: BOOL;
	OP10A_HME_1_5									: INT	:= 5;
	OP10A_HME_5_10									: INT 	:= 10;	
	OP10A_HME_10_15									: INT	:= 15;
	OP10A_HME_15_20									: INT	:= 20;
	OP10A_HME_20_25									: INT	:= 25;
	OP10A_HME_25_30									: INT	:= 30;
	
									(*OP10B*)
	R2												: R_TRIG;									
	OP10B_START_HOMNG								: BOOL;
	OP10B_GRIPPER_HOME								: BOOL;										
	OP10B_ALL_HOME									: BOOL;	
	OP10B_ROBO_SFE_HME								: BOOL;
	OP10B_O_LHGRIP_HMG1								: BOOL;
	OP10B_O_RHGRIP_HMG1								: BOOL;
	OP10B_O_LHPUSH_HMG1								: BOOL;
	OP10B_O_RHPUSH_HMG1								: BOOL;
	OP10B_O_VERT_HMG1								: BOOL;
	OP10B_O_DEGRE_HMG1								: BOOL;
	OP10B_O_HORZ_HMG1								: BOOL;	
	OP10B_GRP_REFERENCED							: BOOL;	
	OP10B_HME_1_5									: INT	:= 5;
	OP10B_HME_5_10									: INT 	:= 10;	
	OP10B_HME_10_15									: INT	:= 15;
	OP10B_HME_15_20									: INT	:= 20;
	OP10B_HME_20_25									: INT	:= 25;
	OP10B_HME_25_30									: INT	:= 30;	

	
// MANUAL

									(*OP10A*)
	OP10A_CYLINDER_ERR								: WORD;	
	OP10A_O_CNVY_JOG_P								: BOOL;
	OP10A_O_CNVY_JOG_N								: BOOL;
	OP10B_O_CNVY_JOG_P								: BOOL;
	OP10B_O_CNVY_JOG_N								: BOOL;
	OP10A_LH_GRP_JOG_P								: BOOL;
	OP10A_LH_GRP_JOG_N								: BOOL;
	OP10A_RH_GRP_JOG_N								: BOOL;
	OP10A_RH_GRP_JOG_P								: BOOL;	
	OP10A_LH_ROTRY_JOG_N							: BOOL;
	OP10A_LH_ROTRY_JOG_P							: BOOL;
	OP10A_RH_ROTRY_JOG_P							: BOOL;
	OP10A_RH_ROTRY_JOG_N							: BOOL;
	OP10A_CYL_PNP_CHECK								: BOOL;
									(*OP10B*)	
	OP10B_CYLINDER_ERR								: WORD;
	OP10B_LH_GRP_JOG_P								: BOOL;
	OP10B_LH_GRP_JOG_N								: BOOL;
	OP10B_RH_GRP_JOG_P								: BOOL;
	OP10B_RH_GRP_JOG_N								: BOOL;
	OP10B_LH_ROTRY_JOG_P							: BOOL;
	OP10B_LH_ROTRY_JOG_N							: BOOL;
	OP10B_RH_ROTRY_JOG_P							: BOOL;
	OP10B_RH_ROTRY_JOG_N							: BOOL;
	OP10_FRST_BDY_GRP_JOG_N							: BOOL;
	OP10_FRST_BDY_GRP_JOG_P							: BOOL;
	OP10_SEC_BDY_GRP_JOG_P							: BOOL;
	OP10_SEC_BDY_GRP_JOG_N							: BOOL;
	OP10B_CYL_PNP_CHECK								: BOOL;
	
// DRY RUN	
	OP10A_DRY_RUN									: BOOL;
	OP10B_Dry_Run									: BOOL;                                            		
// AUTO                                     		
                            (*CYLINDER*)
							  (*OP10*)
	OP10_SRV_ALL_HOME								: BOOL;
	OP10_LH_CMP_RDY_PCK								: BOOL;
	OP10_RH_CMP_RDY_PCK								: BOOL;
	OP10A_SING_CMR_TRIG								: BOOL;
	OP10B_SING_CMR_TRIG								: BOOL;
	OP10A_SING_CAM_DN								: BOOL;
	OP10B_SING_CAM_DN								: BOOL;
							 (*OP10A*)
	OP10A_CYL_RDY_TO_PLC							: BOOL;	
	OP10A_ALL_CYL_HOME_FB							: BOOL;
	OP10A_SRV_ALL_HOME								: BOOL;
	OP10A_O_0DEGRE_AUTOCMD1							: BOOL;
	OP10A_O_180DEGRE_AUTOCMD2						: BOOL;
	OP10A_O_HORZ_AUTOCMD1							: BOOL;
	OP10A_O_HORZ_AUTOCMD2							: BOOL;
	OP10A_A_O_LHGRIP_ONOFF							: BOOL;
	OP10A_A_O_LHPUSH_CYL							: BOOL;
	OP10A_A_LH_REJ_HOME								: BOOL;
	OP10A_A_LH_REJ_WRK								: BOOL;
	OP10A_A_O_RHGRIP_ONOFF							: BOOL;
	OP10A_A_O_RHPUSH_CYL							: BOOL;
	OP10A_A_RH_REJ_HOME								: BOOL;
	OP10A_A_RH_REJ_WRK								: BOOL;
	OP10A_O_VERT_AUTOCMD1							: BOOL;
	OP10A_O_VERT_AUTOCMD2							: BOOL;
	OP10A_BDY1_PCK_BYPAS							: BOOL;
	OP10A_BDY2_PCK_BYPAS							: BOOL;
	OP10A_ORNG_RDY_PCK								: BOOL;
	OP10A_ORNG_PCK_DN								: BOOL;
							 (*OP10B*)
	OP10B_CYL_RDY_TO_PLC							: BOOL;
	OP10B_ALL_CYL_HOME_FB							: BOOL;
	OP10B_SRV_ALL_HOME								: BOOL;
	OP10B_O_0DEGRE_AUTOCMD1							: BOOL;
	OP10B_O_180DEGRE_AUTOCMD2						: BOOL;
	OP10B_O_HORZ_AUTOCMD1							: BOOL;
	OP10B_O_HORZ_AUTOCMD2							: BOOL;
	OP10B_A_O_LHGRIP_ONOFF							: BOOL;
	OP10B_A_O_LHPUSH_CYL							: BOOL;
	OP10B_A_LH_REJ_HOME								: BOOL;
	OP10B_A_LH_REJ_WRK								: BOOL;
	OP10B_A_O_RHGRIP_ONOFF							: BOOL;
	OP10B_A_O_RHPUSH_CYL							: BOOL;
	OP10B_A_RH_REJ_HOME								: BOOL;
	OP10B_A_RH_REJ_WRK								: BOOL;
	OP10B_O_VERT_AUTOCMD1							: BOOL;
	OP10B_O_VERT_AUTOCMD2							: BOOL;
	OP10B_BDY1_PCK_BYPAS							: BOOL;
	OP10B_BDY2_PCK_BYPAS							: BOOL;
	OP10B_ORNG_RDY_PCK								: BOOL;
	OP10B_ORNG_PCK_DN								: BOOL;  

	
// CAMERA
								(*OP10A_CAMERA*)		
	OP10A_CMR_DN_RSLT								: BOOL;
	OP10A_LH_CMR_OK									: BOOL;
	OP10A_LH_CMR_NOK								: BOOL;	
	OP10A_RH_CMR_OK									: BOOL;
	OP10A_RH_CMR_NOK								: BOOL;	
								(*OP10B_CAMERA*)		
	OP10B_CMR_DN_RSLT								: BOOL;
	OP10B_LH_CMR_OK									: BOOL;
	OP10B_LH_CMR_NOK								: BOOL;	
	OP10B_RH_CMR_OK									: BOOL;
	OP10B_RH_CMR_NOK								: BOOL;	
	
	
	
	
	
// WILL BE DELETED
	OP10A_MODE_BLOCK: Mode_Selection_Block1;
	OP10A_MODE_WORD: INT;
	OP10A_AUTO_SELECTED: BOOL;
	OP10A_MANUAL_SELECTED: BOOL;
	OP10A_STEP_SELECTED: BOOL;
	OP10A_AUTO_RUNNING: BOOL;
	OP10A_STEP_RUNNING: BOOL;
	OP10A_START_ENABLE: BOOL;
	OP10A_MACHINE_STOP: BOOL;
	OP10A_ERR: BOOL;

	OP10B_MODE_BLOCK: Mode_Selection_Block1;
	OP10B_MODE_WORD: INT;
	OP10B_AUTO_SELECTED: BOOL;
	OP10B_MANUAL_SELECTED: BOOL;
	OP10B_STEP_SELECTED: BOOL;
	OP10B_AUTO_RUNNING: BOOL;
	OP10B_STEP_RUNNING: BOOL;
	OP10B_START_ENABLE: BOOL;
	OP10B_MACHINE_STOP: BOOL;
	OP10B_ERR: BOOL; 

	
	CHECK				: BOOL;
	
	
//Camera GVLs
	OP10A_LH_Camera_Trigger		      : BOOL;
	OP10A_LH_Camera_Job_Change_start   : BOOL;
	OP10A_LH_Camera_Error			  : BOOL;
	OP10A_LH_Camera_Ready			  : BOOL;
	OP10A_LH_Camera_Online			  : BOOL;	
	OP10A_LH_Job_Change_Complete		    : BOOL;
	OP10A_LH_Job_Change_Error   		    : BOOL;
	OP10A_LH_Picture_Taken      		    : BOOL;
	OP10A_LH_Error_status				: STRING;
	OP10A_LH_Target_Job_ID				: UINT;
	OP10A_LH_Loaded_Job_ID		    	: UINT;

	OP10A_RH_Camera_Trigger		      : BOOL;
	OP10A_RH_Camera_Job_Change_start   : BOOL;
	OP10A_RH_Camera_Error			  : BOOL;
	OP10A_RH_Camera_Ready			  : BOOL;
	OP10A_RH_Camera_Online			  : BOOL;	
	OP10A_RH_Job_Change_Complete		: BOOL;
	OP10A_RH_Job_Change_Error   		: BOOL;
	OP10A_RH_Picture_Taken      		: BOOL;
	OP10A_RH_Error_status				: STRING;
	OP10A_RH_Target_Job_ID				: UINT;
	OP10A_RH_Loaded_Job_ID		    	: UINT;

	OP10B_LH_Camera_Trigger		      : BOOL;
	OP10B_LH_Camera_Job_Change_start   : BOOL;
	OP10B_LH_Camera_Error			  : BOOL;
	OP10B_LH_Camera_Ready			  : BOOL;
	OP10B_LH_Camera_Online			  : BOOL;	
	OP10B_LH_Job_Change_Complete		    : BOOL;
	OP10B_LH_Job_Change_Error   		    : BOOL;
	OP10B_LH_Picture_Taken      		    : BOOL;
	OP10B_LH_Error_status				: STRING;
	OP10B_LH_Target_Job_ID				: UINT;
	OP10B_LH_Loaded_Job_ID		    	: UINT;

	OP10B_RH_Camera_Trigger		      : BOOL;
	OP10B_RH_Camera_Job_Change_start   : BOOL;
	OP10B_RH_Camera_Error			  : BOOL;
	OP10B_RH_Camera_Ready			  : BOOL;
	OP10B_RH_Camera_Online			  : BOOL;	
	OP10B_RH_Job_Change_Complete		    : BOOL;
	OP10B_RH_Job_Change_Error   		    : BOOL;
	OP10B_RH_Picture_Taken      		    : BOOL;
	OP10B_RH_Error_status				: STRING;
	OP10B_RH_Target_Job_ID				: UINT;
	OP10B_RH_Loaded_Job_ID		    	: UINT;

	OP10A_Camera_Trigger_Ack: BOOL;
	OP10A_Miss_Trigger: BOOL;
	OP10A_LH_Camera_OK  : BOOL;
	OP10A_LH_Camera_NOK : BOOL;
	OP10A_RH_Camera_OK  : BOOL;
	OP10A_RH_Camera_NOK : BOOL;
	OP10A_Camera_Done	: BOOL;
	
	OP10B_Camera_Trigger_Ack: BOOL;
	OP10B_Miss_Trigger: BOOL;
	OP10B_LH_Camera_OK  : BOOL;
	OP10B_LH_Camera_NOK : BOOL;
	OP10B_RH_Camera_OK  : BOOL;
	OP10B_RH_Camera_NOK : BOOL;
	OP10B_Camera_Done	: BOOL;	
	
	Conv_Step_no_10A: INT;
	Conv_Step_no_10B: INT;
	
//Empty Camera
	OP10A_Empty_Cam_1_Camera_Trigger		    : BOOL;
	OP10A_Empty_Cam_1_Camera_Job_Change_start   : BOOL;
	OP10A_Empty_Cam_1_Camera_Error			  : BOOL;
	OP10A_Empty_Cam_1_Camera_Ready			  : BOOL;
	OP10A_Empty_Cam_1_Camera_Online			  : BOOL;	
	
	OP10B_Empty_Cam_2_Camera_Trigger		    : BOOL;
	OP10B_Empty_Cam_2_Camera_Job_Change_start   : BOOL;
	OP10B_Empty_Cam_2_Camera_Error			  : BOOL;
	OP10B_Empty_Cam_2_Camera_Ready			  : BOOL;
	OP10B_Empty_Cam_2_Camera_Online			  : BOOL;

	OP10A_Body_OK			 :BOOL; 
	OP10A_Body_NOK			 :BOOL; 
	OP10A_Body_Window_0Deg	 :BOOL; 
	OP10A_Body_Window_90Deg	 :BOOL;	
	OP10B_Body_OK			 :Bool; 
	OP10B_Body_NOK			 :Bool;  
	OP10B_Body_Window_0Deg	 :BOOL; 
	OP10B_Body_Window_90Deg	 :BOOL; 
	
	OP10A_Pick_Ready		 :BOOL;
	OP10A_Pick_Done			 :BOOL;
	
	OP10B_Pick_Ready		 :BOOL;
	OP10B_Pick_Done			 :BOOL;	
	
	OP10A_Sing_Seq  : INT;//Singulation Sequence
	OP10B_Sing_Seq  : INT;	
END_VAR

VAR_GLOBAL PERSISTENT

	OP10_COMP_PICKED_1						: BOOL;
	OP10_COMP_PICKED_2						: BOOL;
	OP10A_SING_CAM_BYPASS					: BOOL;
	OP10B_SING_CAM_BYPASS					: BOOL;
//Drum_Feeder
	OP10A_Drum_Feed_Motor_Speed		AT %Q*  : INT;	
	OP10A_HMI_Drum_Feed_Mtr_Speed_IP		: INT;
	OP10A_Drum_Feed_Mtr_Speed_Select		: BOOL;
	OP10A_Drum_Feed_Mtr_Run_Fwd 			: BOOL;
	OP10A_Drum_Feed_Mtr_Reset   			: BOOL;
	
//Drum_Feeder
	OP10B_Drum_Feed_Motor_Speed		AT %Q*  : INT;	
	OP10B_HMI_Drum_Feed_Mtr_Speed_IP		: INT;
	OP10B_Drum_Feed_Mtr_Speed_Select		: BOOL;
	OP10B_Drum_Feed_Mtr_Run_Fwd 			: BOOL;
	OP10B_Drum_Feed_Mtr_Reset   			: BOOL;	
	
	OP10A_Conv_Fwd_Time_6_3			: INT:=750;
	OP10A_Conv_Fwd_Speed_6_3		: INT:=150;
	OP10A_Conv_Rev_Time_6_3			: INT:=500;
	OP10A_Conv_Rev_Speed_6_3		: INT:=-100;     
	OP10A_Conv_Fwd_Time_7_89		: INT:=750;
	OP10A_Conv_Fwd_Speed_7_89		: INT:=150;
	OP10A_Conv_Rev_Time_7_89		: INT:=500;
	OP10A_Conv_Rev_Speed_7_89		: INT:=-100;			  
	OP10A_Conveyor_Speed			: REAL;
	OP10A_Model						: STRING[80];	

	OP10B_Conv_Fwd_Time_6_3			: INT:=750;
	OP10B_Conv_Fwd_Speed_6_3		: INT:=150;
	OP10B_Conv_Rev_Time_6_3			: INT:=500;
	OP10B_Conv_Rev_Speed_6_3		: INT:=-100;     
	OP10B_Conv_Fwd_Time_7_89		: INT:=750;
	OP10B_Conv_Fwd_Speed_7_89		: INT:=150;
	OP10B_Conv_Rev_Time_7_89		: INT:=500;
	OP10B_Conv_Rev_Speed_7_89		: INT:=-100;			  
	OP10B_Conveyor_Speed			: REAL;
	OP10B_Model						: STRING[80];	

END_VAR

// ---- POUs/Programs/OP120/OP120_GVL.TcGVL

VAR_GLOBAL
	//GENERAL
OP120_Auto:					BOOL;
OP120_HomeRunning:			BOOL;
OP120_ErrorActive:			BOOL;
OP120_Home_PB:				BOOL;
OP120_Work_PB:				BOOL;
OP120_ManualSafetyBypass:	BOOL;
OP120_LightCurtainBypass:	BOOL;
OP120_OperationCompleted:	BOOL;
OP120_LampCheck:			BOOL;
OP120_MachineLamp:			BOOL;
OP120_ComponentOk:			BOOL;
OP120_ComponentNok:			BOOL;
OP120_RepeatBit:			BOOL;
OP120_HomingResetBit:		BOOL;
OP120_ControlledByRobo:		BOOL;
OP120_Any_Bypass:			BOOL;
OP120_ManualModeStatus:		INT;
OP120_ManualModeWord:		INT;
OP120_STN_MOVER				: INT;
OP120Seq:				INT;
OP120_LH_AutoSeq: 			INT;
OP120_RH_AutoSeq: 			INT;
OP120_Homing_Seq:			INT;

Automatic_Run:				BOOL;
OP120_Prev_Stat_Operation_Completed: BOOL;
OP120_Prev_Comp_Status: INT;
OP120_Prev_LH_COMP_OK:BOOL;
OP120_Prev_LH_COMP_NOK:BOOL;
OP120_Prev_RH_COMP_OK:BOOL;
OP120_Prev_RH_COMP_NOK:BOOL;
OP120_LH_Operation_Completed:BOOL;
OP120_RH_Operation_Completed:BOOL;

OP120_LH_Comp_OK: BOOL;
OP120_LH_Comp_NOK: BOOL;
OP120_RH_Comp_OK: BOOL;
OP120_RH_Comp_NOK: BOOL;

OP120_RH_Laser_Start:BOOL;
OP120_LH_Laser_Start:BOOL;
OP120_RH_Laser_Completed:BOOL;
OP120_LH_Laser_Completed:BOOL;
OP120_Comp_Picked:BOOL;


//AutoSequence 
OP120_AutoSeq:			INT;

//ModeSelection Outputs
//OP120_AutoSelected:		    BOOL;
OP120_ManualSelected:		BOOL;
OP120_StepSelected:			BOOL;
OP120_AutoSelected:		    BOOL;
OP120_AutoRunning :BOOL;
OP120_StepRunning:BOOL;
OP120_StartEnable:BOOL;
OP120_Machine_Stop:BOOL;
//MAnual Control Tags
CR120_Lifting_Cyl: Cylinder_Block;
 CR120_Horizontal_Push_Cyl: Cylinder_Block;
 CR120_Camera_Slide_Cyl: Cylinder_Block;
CR120_Gripper_Cyl: Cylinder_Block;
	SR120_Oring_Feed_Servo: FB_Axis;
	SR120_Oring_Feed_Servo_Axis:AXIS_REF;
	SR120_Oring_Feed_Servo_Control:Servo_Control;
	SR120_Oring_Feed_Manual_Axis:stManualModeAxis;


//Manual Cylinder FB Tags
OP120_Lifting_Cyl_Status:	 INT;
OP120_Gripper_Cyl_Status:	 INT;
OP120_Horizontal_Push_Cyl_Status:INT;
OP120_Camera_Slide_Cyl_Status:INT;
//HMI Tags(From HMI)
OP120_HMI_AutoMode:						BOOL;
OP120_HMI_ManualMOde:					BOOL;
OP120_HMI_StepMode:						BOOL;
OP120_HMI_CycleStart_PB:				BOOL;
OP120_HMI_Homing_PB:					BOOL;
CR120_HMI_Gripper_Cyl_Home_PB:			BOOL;
CR120_HMI_Gripper_Cyl_Work_PB:			BOOL;
CR120_HMI_Lifting_Cyl_Home_PB:			BOOL;
CR120_HMI_Lifting_Cyl_Work_PB:			BOOL;
CR120_HMI_Horizontal_Push_Cyl_Home_PB:	BOOL;
CR120_HMI_Horizontal_Push_Cyl_Work_PB:	BOOL;
CR120_HMI_Camera_Slide_Cyl_Home_PB:	BOOL;
CR120_HMI_Camera_Slide_Cyl_Work_PB:	BOOL;
OP120_HMI_Bowl_ON_Time:					TIME;
OP120_HMI_Bowl_OFF_time:				TIME;
OP120_HMI_Bowl_On_PB:					BOOL;
OP120_HMI_Hopper_On_PB:					BOOL;
OP120_HMI_Reset:						BOOL;
//Error
OP120_ErrorWord_0:    							 DINT;
OP120_ErrorWord_1:								 DINT;
OP120_ErrorWord_2:								 DINT;

// Robo Inouts
OP120_Ready_To_Pick:					BOOL;
OP120_Lring_Placed:						BOOL;

//Camera Inputs
OP120_Camera_OK:								BOOL;
OP120_Camera_NOK:								BOOL;
OP120_Robo_ProgramReset: BOOL;

	OP120_Temp_Home_OK: BOOL;
	OP120_HomeCondition_OK: BOOL;
	OP120_OperationEnable: BOOL;
	OP130_CycleTime: UDINT;
	b1sec: BOOL;
//Robo Seq Inputs

CheckParkOK: BOOL;
CheckParkNOK: BOOL;
OP120_PushPlace:BOOL;
Part_Picked: BOOL;
Ready_for_next_singulation:BOOL;
OP120_PartPushed: BOOL;
Op120_PartPlaced:BOOL;
OP120_Sing_AutoSeq:INT;
OP120_Lock_AutoSeq:INT;
OP120_Bowl_OK:BOOL;
OP120_Camera_Auto_Trigger: BOOL;
OP120_CamOK: BOOL;
pickParkOK: BOOL;
pickParkNOK: BOOL;
OP120_CamNOK: BOOL;
OP120_MoverinStation:BOOL;
OP120_MoverPresent:BOOL;
tempdelete1:BOOL;
TempDelete3:BOOL;
Op120_DryrunOK:BOOL;
Op120_Bowl_SeqRun:BOOL;

OP120_Vaccuum_IP_Port5_Byte1 AT %I* : BYTE;
OP120_Vaccuum_IP_Port5_Byte2 AT %I* : BYTE;
OP120_Vaccuum_OP_Port5_Byte1 AT %Q* : BYTE;
OP120_Vaccuum_OP_Port5_Byte2 AT %Q* : BYTE;

OP120_Vaccuum_IP_Port6_Byte1 AT %I* : BYTE;
OP120_Vaccuum_IP_Port6_Byte2 AT %I* : BYTE;
OP120_Vaccuum_OP_Port6_Byte1 AT %Q* : BYTE;
OP120_Vaccuum_OP_Port6_Byte2 AT %Q* : BYTE;

OP120_Vaccum1_Bit0 :BOOL;
OP120_Vaccum1_Bit1 :BOOL;
OP120_Vaccum2_Bit0 :BOOL;
OP120_Vaccum2_Bit1 :BOOL;

OP120_GotoPick :BOOL;
OP120_STN_ENABLE: BOOL;
Op120_PartSingulated: BOOL;

// temp need to be deleted
temp_var : ARRAY [0..1000] OF BOOL;


conveyor_status :INT;
robot_status    :INT;	

	
	op120_setuserdata: BOOL;
	op120_all_camera_ok: BOOL;
END_VAR
VAR_GLOBAL PERSISTENT
	
	op120_modelselected: INT;
END_VAR

// ---- POUs/Programs/OP120/OP120_IO_Tag_Link.TcGVL

VAR_GLOBAL
	


	
	
//Robot Inputs
OP120_SO_Mirror_Auto_enable AT %I*:BOOL;
OP120_SO_Program_Execute AT %I*:BOOL;
OP120_SO_Program_Waiting AT %I*:BOOL;
OP120_SO_Program_Waiting2 AT %I*:BOOL;
OP120_SO_Stop_Status AT %I*:BOOL;
OP120_SO_Program_Sel_enabled_OP AT %I*:BOOL;
OP120_SO_During_error AT %I*:BOOL;
OP120_SO_During_Cycle_Stop AT %I*:BOOL;
OP120_SO_Mirror_SRVO_Off AT %I*:BOOL;
OP120_SO_Servo_ON_OFF_Status AT %I*:BOOL;
OP120_SO_Auto_Operation_Enable AT %I*:BOOL;
OP120_SO_Moving_Home AT %I*:BOOL;
OP120_SO_Spare1 AT %I*:BOOL;
OP120_SO_During_Machine_Lock AT %I*:BOOL;
OP120_SO_H_Error AT %I*:BOOL;
OP120_SO_L_Error AT %I*:BOOL;
OP120_SO_Caution AT %I*:BOOL;
OP120_SO_During_EMG_Stop AT %I*:BOOL;
OP120_SO_Teach_Mode AT %I*:BOOL;
OP120_SO_Auto_OP_Mode AT %I*:BOOL;
OP120_SO_Auto_Ext_Mode AT %I*:BOOL;
OP120_SO_TP_Enable AT %I*:BOOL;
OP120_SO_Heartbeat AT %I*:BOOL;
OP120_SO_Spare2 AT %I*:BOOL;
OP120_SO_Rbt_In_Home AT %I*:BOOL;
OP120_SO_Rbt_In_Pick_Zone AT %I*:BOOL;
OP120_SO_Rbt_In_Place_Zone AT %I*:BOOL;
OP120_SO_Rbt_In_Reject_Zone AT %I*:BOOL;
OP120_SO_Rbt_In_ATC_Zone AT %I*:BOOL;
OP120_SO_Spare4 AT %I*:BOOL;
OP120_SO_Spare5 AT %I*:BOOL;
OP120_SO_Spare6 AT %I*:BOOL;

OP120_GO_Mode_Ack AT %I*:BYTE;
OP120_GO_Variant_number_Ack AT %I*:BYTE;
OP120_GO_Position_Rchd_Ack AT %I*:BYTE;
OP120_GO_Auto_Status AT %I*:BYTE;
OP120_GO_Byte_Spare1 AT %I*:BYTE;
OP120_GO_Byte_Spare2 AT %I*:BYTE;
OP120_GO_Byte_Spare3 AT %I*:BYTE;
OP120_GO_Byte_Spare4 AT %I*:BYTE;
OP120_GO_Error_Number AT %I*:BYTE;
OP120_GO_Word_Spare AT %I*:BYTE;


OP120_EO_Sequence_Running AT %I*:BOOL;
OP120_EO_Sequence_Completed AT %I*:BOOL;
OP120_EO_Spring_Pick_Completed AT %I*:BOOL;
OP120_EO_Spring_Place_Pos_Reached AT %I*:BOOL;
OP120_EO_Spring_Place_Completed AT %I*:BOOL;
OP120_EO_NOK_Part_Dropped AT %I*:BOOL;
OP120_EO_Spare2 AT %I*:BOOL;
OP120_EO_Spare3 AT %I*:BOOL;
OP120_EO_Spare4 AT %I*:BOOL;
OP120_EO_Spare5 AT %I*:BOOL;
OP120_EO_Spare6 AT %I*:BOOL;
OP120_EO_Spare7 AT %I*:BOOL;
OP120_EO_Spare8 AT %I*:BOOL;
OP120_EO_Spare9 AT %I*:BOOL;
OP120_EO_Step_Reached AT %I*:BOOL;
OP120_EO_Spare11 AT %I*:BOOL;
OP120_EO_RO_Gripper1_Open AT %I*:BOOL;
OP120_EO_RO_Gripper1_Close AT %I*:BOOL;
OP120_EO_RO_Gripper2_Open AT %I*:BOOL;
OP120_EO_RO_Gripper2_Close AT %I*:BOOL;
OP120_EO_RO_ATC_Open AT %I*:BOOL;
OP120_EO_RO_ATC_Close AT %I*:BOOL;
OP120_EO_RO_Spare18 AT %I*:BOOL;
OP120_EO_RO_Spare19 AT %I*:BOOL;
OP120_EO_RI_Gripper1_Open_FB AT %I*:BOOL;
OP120_EO_RI_Gripper1_Close_FB AT %I*:BOOL;
OP120_EO_RI_Gripper2_Open_FB AT %I*:BOOL;
OP120_EO_RI_Gripper2_Close_FB AT %I*:BOOL;
OP120_EO_RI_ATC_Open_FB AT %I*:BOOL;
OP120_EO_RI_ATC_Close_FB AT %I*:BOOL;
OP120_EO_ATC_Tool_Presence_1 AT %I*:BOOL;
OP120_EO_ATC_Tool_Presence_2 AT %I*:BOOL;

//Robo Outputs
OP120_SI_Auto_Enable AT %Q*:BOOL;
OP120_SI_Start AT %Q*:BOOL;
OP120_SI_Stop AT %Q*:BOOL;
OP120_SI_Stop2 AT %Q*:BOOL;
OP120_SI_Spare1 AT %Q*:BOOL;
OP120_SI_Program_Reset AT %Q*:BOOL;
OP120_SI_Error_Reset AT %Q*:BOOL;
OP120_SI_Cycle_Stop AT %Q*:BOOL;
OP120_SI_Servo_OFF AT %Q*:BOOL;
OP120_SI_Servo_ON AT %Q*:BOOL;
OP120_SI_Operation_Enable AT %Q*:BOOL;
OP120_SI_Move_Home AT %Q*:BOOL;
OP120_SI_General_Output_reset AT %Q*:BOOL;
OP120_SI_Machine_Lock AT %Q*:BOOL;
OP120_SI_Spare2 AT %Q*:BOOL;
OP120_SI_Spare3 AT %Q*:BOOL;
OP120_SI_Spare4 AT %Q*:BOOL;
OP120_SI_Spare5 AT %Q*:BOOL;
OP120_SI_Spare6 AT %Q*:BOOL;
OP120_SI_Spare7 AT %Q*:BOOL;
OP120_SI_Spare8 AT %Q*:BOOL;
OP120_SI_Spare9 AT %Q*:BOOL;
OP120_SI_PLC_Heartbeat AT %Q*:BOOL;
OP120_SI_Dry_Run AT %Q*:BOOL;
OP120_SI_Homing_Start AT %Q*:BOOL;
OP120_SI_Pick_Zone_Safe AT %Q*:BOOL;
OP120_SI_Place_Zone_Safe AT %Q*:BOOL;
OP120_SI_Reject_Zone_Safe AT %Q*:BOOL;
OP120_SI_ATC_Tool_Safe AT %Q*:BOOL;
OP120_SI_Spare11 AT %Q*:BOOL;
OP120_SI_Spare12  AT %Q*:BOOL;
OP120_SI_Spare13 AT %Q*:BOOL;


OP120_GI_Mode AT %Q*:BYTE;
OP120_GI_Variant_number AT %Q*:BYTE;
OP120_GI_Position_Number AT %Q*:BYTE;
OP120_GI_Byte_Spare1 AT %Q*:BYTE;
OP120_GI_Byte_Spare2  AT %Q*:BYTE;
OP120_GI_Byte_Spare3 AT %Q*:BYTE;
OP120_GI_Byte_Spare4 AT %Q*:BYTE;
OP120_GI_Byte_Spare5 AT %Q*:BYTE;
OP120_GI_Word_Spare AT %Q*:BYTE;
OP120_GI_Word_Spare1 AT %Q*:BYTE;

OP120_EI_Manual_Seq_Start AT%Q*:BOOL;
OP120_EI_Spare2 AT%Q*:BOOL;
OP120_EI_Rdy_Pick_Spring AT%Q*:BOOL;
OP120_EI_Rdy_Place_Spring AT%Q*:BOOL;
OP120_EI_Insertion_Complete AT%Q*:BOOL;
OP120_EI_Rdy_Place_Rejection AT%Q*:BOOL;
OP120_EI_Spare4 AT%Q*:BOOL;
OP120_EI_Spare5 AT%Q*:BOOL;
OP120_EI_Spare6 AT%Q*:BOOL;
OP120_EI_Spare7 AT%Q*:BOOL;
OP120_EI_Spare8 AT%Q*:BOOL;
OP120_EI_Spare9 AT%Q*:BOOL;
OP120_EI_Spare10 AT%Q*:BOOL;
OP120_EI_Spare11 AT%Q*:BOOL;
OP120_EI_Step_Continue AT%Q*:BOOL;
OP120_EI_Spare13 AT%Q*:BOOL;
OP120_EI_Gripper1_Open AT%Q*:BOOL;
OP120_EI_Gripper1_Close AT%Q*:BOOL;
OP120_EI_Gripper2_Open AT%Q*:BOOL;
OP120_EI_Gripper2_Close AT%Q*:BOOL;
OP120_EI_ATC_Open AT%Q*:BOOL;
OP120_EI_ATC_Close AT%Q*:BOOL;
OP120_EI_Spare21 AT%Q*:BOOL;
OP120_EI_Spare22 AT%Q*:BOOL;
OP120_EI_Spare23 AT%Q*:BOOL;
OP120_EI_Spare24 AT%Q*:BOOL;
OP120_EI_Spare25 AT%Q*:BOOL;
OP120_EI_Spare26 AT%Q*:BOOL;
OP120_EI_Spare27 AT%Q*:BOOL;
OP120_EI_Spare28 AT%Q*:BOOL;
OP120_EI_Spare29 AT%Q*:BOOL;
OP120_EI_Spare30 AT%Q*:BOOL;


//Registerin
OP120_Robo_In6001 AT%I*:UINT;
OP120_Robo_In6002 AT%I*:UINT;
OP120_Robo_In6003 AT%I*:UINT;
OP120_Robo_In6004 AT%I*:UINT;
OP120_Robo_In6005 AT%I*:UINT;
OP120_Robo_In6006 AT%I*:UINT;
OP120_Robo_In6007 AT%I*:UINT;
OP120_Robo_In6008 AT%I*:UINT;
OP120_Robo_In6009 AT%I*:UINT;
OP120_Robo_In6010 AT%I*:UINT;
OP120_Robo_In6011 AT%I*:UINT;
OP120_Robo_In6012 AT%I*:UINT;

OP120_Robo_Out6001 AT%Q*:UINT;
OP120_Robo_Out6002 AT%Q*:UINT;
OP120_Robo_Out6003 AT%Q*:UINT;
OP120_Robo_Out6004 AT%Q*:UINT;
OP120_Robo_Out6005 AT%Q*:UINT;
OP120_Robo_Out6006 AT%Q*:UINT;
OP120_Robo_Out6007 AT%Q*:UINT;
OP120_Robo_Out6008 AT%Q*:UINT;
OP120_Robo_Out6009 AT%Q*:UINT;
OP120_Robo_Out6010 AT%Q*:UINT;


END_VAR

// ---- POUs/Programs/XTS/HMI_GVL.TcGVL
//{attribute 'qualified_only'}
VAR_GLOBAL
		
END_VAR
VAR_GLOBAL PERSISTENT
	ZERO_POS_NO								: INT :=1;
	OP10A_XTS_POS_NO						: INT;
	OP10B_XTS_POS_NO						: INT;
	OP20_XTS_POS_NO					        : INT;
	OP30_XTS_POS_NO                         : INT;
	OP40_XTS_POS_NO                         : INT;
	OP50_XTS_POS_NO                         : INT;
	OP60_XTS_POS_NO                         : INT;
	OP70_XTS_POS_NO                         : INT;
	OP80_XTS_POS_NO                         : INT;
	OP90_XTS_POS_NO                         : INT;
	OP110_XTS_POS_NO                        : INT;
	OP120_XTS_POS_NO                        : INT;
	OP130_XTS_POS_NO                        : INT;
	OP140_XTS_POS_NO                     	: INT;
	OP140_P1_XTS_POS_NO                    	: INT;	
	OP140_P2_XTS_POS_NO                    	: INT;	
	OP140_P3_XTS_POS_NO                    	: INT;	
	OP150A_LH_XTS_POS_NO					: INT;
	OP150A_RH_XTS_POS_NO					: INT;
	OP150B_LH_XTS_POS_NO					: INT;
	OP150B_RH_XTS_POS_NO					: INT;
	OP150C_LH_XTS_POS_NO					: INT;
	OP150C_RH_XTS_POS_NO					: INT;		
	OP160_XTS_POS_NO                        : INT;
	AUTO_WITH_XTS							: BOOL;
	
	
END_VAR

// ---- POUs/Programs/XTS/XTS_GVL.TcGVL
//{attribute 'qualified_only'}
VAR_GLOBAL
	MOVER_POS_RECHED						: ARRAY [0..nNumberofMovers] OF BOOL;
	MOVER_POSITION							: ARRAY[0..nNumberOfStations]OF INT;
	nCAGroupState							: INT;
	OP130_MVR_DN_PERMISSION					: BOOL;	
	STATION_DONE							: ARRAY[0..nNumberofMovers] OF ARRAY[0..nNumberOfStations]OF BOOL;														
END_VAR
VAR_GLOBAL PERSISTENT
	MOVER_CMP_STATUS						: ARRAY [0..nNumberofMovers] OF ARRAY [1..3] OF INT;
	XTS_STOP_POSITION						: ARRAY[1..nNumberOfStations] OF LREAL;
	MOVER_STP_NO							: ARRAY [0..nNumberofMovers] OF INT;
END_VAR

// ---- GVLs/GVL.TcGVL
{attribute 'qualified_only'}
VAR_GLOBAL
	EC_MasterNetID_Arr_X1 	AT %I*:	T_AmsNetIdArr;
	EC_MasterNetID_Arr_X2   AT %I*:	T_AmsNetIdArr;
	EC_MasterNetID_Arr_X3   AT %I*:	T_AmsNetIdArr;
	
	bExecute			: BOOL;
	nNoOf_Cfg_Slaves	: UINT;
	nNoOf_Slaves_Read	: UINT;

END_VAR
VAR_GLOBAL CONSTANT
	ECAT_MAX_SLAVES_X1: INT := 80;
	ECAT_MAX_SLAVES_X2: INT := 30;
	ECAT_MAX_SLAVES_X3: INT := 50;
END_VAR

// ---- GVLs/RayPRO_Variables.TcGVL

VAR_GLOBAL
	
	{attribute 'OPC.UA.DA':='1'}
	StatusMachineOn			 	: BOOL;
	{attribute 'OPC.UA.DA':='1'}
	StatusToolChange         	: BOOL;
	{attribute 'OPC.UA.DA':='1'}
	StatusSettings           	: BOOL;
	{attribute 'OPC.UA.DA':='1'}
	StatusProducingParts     	: BOOL;
	{attribute 'OPC.UA.DA':='1'}
	StatusStop               	: BOOL;
	{attribute 'OPC.UA.DA':='1'}
	StatusEmptying           	: BOOL;
	{attribute 'OPC.UA.DA':='1'}
	StatusEmpty              	: BOOL;
	{attribute 'OPC.UA.DA':='1'}
	PLCAliveCounter  		 	: DINT;
	{attribute 'OPC.UA.DA':='1'}
	PLCTimeSync		 		 	: DINT;
	{attribute 'OPC.UA.DA':='1'}
	PLCStopRequestAck 		 	: DINT;
	{attribute 'OPC.UA.DA':='1'}
	PLCStoppageSync             : DINT;
	{attribute 'OPC.UA.DA':='1'}
	CurrentStopId				: DINT;
	{attribute 'OPC.UA.DA':='1'}
	CurrentStopHourOfStartTime  : DINT;
	{attribute 'OPC.UA.DA':='1'}
	CurrentStopMinuteOfStartTime: DINT;
	{attribute 'OPC.UA.DA':='1'}
	CurrentStopSecondOfStartTime: DINT;
	{attribute 'OPC.UA.DA':='1'}
	CurrentStopStation			: DINT;
	{attribute 'OPC.UA.DA':='1'}
	CurrentStopCause			: DINT;
	{attribute 'OPC.UA.DA':='1'}
	PLCChangeOfbatchStatus		: DINT;
	{attribute 'OPC.UA.DA':='1'}
	BatchMarking				: STRING;
	{attribute 'OPC.UA.DA':='1'}
	PLCSyncSetup				: DINT;
	{attribute 'OPC.UA.DA':='1'}
	BatchGoodPartQuantity		: DINT;
	{attribute 'OPC.UA.DA':='1'}
	BatchScrappedQuantity		: DINT;
	{attribute 'OPC.UA.DA':='1'}
	BatchDefectCounter1			: DINT;
	{attribute 'OPC.UA.DA':='1'}
	BatchDefectCounter2			: DINT;
	{attribute 'OPC.UA.DA':='1'}
	FirstSamplingStatus			: DINT;
	{attribute 'OPC.UA.DA':='1'}
	PeriodicSamplingStatus		: DINT;
	{attribute 'OPC.UA.DA':='1'}
	ManualSamplingStatus		: DINT;
	{attribute 'OPC.UA.DA':='1'}
	CleanedPartSamplingQuantity	: DINT;
	{attribute 'OPC.UA.DA':='1'}
	CleanedPartSamplingRequest	: DINT;
	{attribute 'OPC.UA.DA':='1'}
	LastSamplingStatus			: DINT;	
	
///MES TAGS
	
	{attribute 'OPC.UA.DA':='1'}
	MESAliveCounter				: DINT;
	{attribute 'OPC.UA.DA':='1'}
	HourOfTime					: DINT;
	{attribute 'OPC.UA.DA':='1'}
	MinuteOfTime        		: DINT;
	{attribute 'OPC.UA.DA':='1'}
	SecondOfTime        		: DINT;
	{attribute 'OPC.UA.DA':='1'}
	TimeOffset          		: DINT;
	{attribute 'OPC.UA.DA':='1'}
	MESStopRequestCounter  		: DINT;
	{attribute 'OPC.UA.DA':='1'}
	MESStoppageSync        		: DINT;
	{attribute 'OPC.UA.DA':='1'}
	MESChangeOfBatchRequest 	: BOOl;
	{attribute 'OPC.UA.DA':='1'}
	IsProductMarked				: BOOl;
	{attribute 'OPC.UA.DA':='1'}
	MarkingCommentLine1			: STRING;
	{attribute 'OPC.UA.DA':='1'}
	MarkingCommentLine2			: STRING;
	{attribute 'OPC.UA.DA':='1'}
	MESSyncSetup				: DINT;
	{attribute 'OPC.UA.DA':='1'}
	HandlingUnitSize			: DINT;
	{attribute 'OPC.UA.DA':='1'}
	FirstSamplingQuantity		: DINT;
	{attribute 'OPC.UA.DA':='1'}
	FirstSamplingRequest		: DINT;
	{attribute 'OPC.UA.DA':='1'}
	FirstSamplingAck			: DINT;
	{attribute 'OPC.UA.DA':='1'}
	PeriodicSamplingQuantity    : DINT;
	{attribute 'OPC.UA.DA':='1'}
	PeriodicSamplingAck         : DINT;
	{attribute 'OPC.UA.DA':='1'}
	ManualSamplingQuantity      : DINT;
	{attribute 'OPC.UA.DA':='1'}
	ManualSamplingRequest       : DINT;
	{attribute 'OPC.UA.DA':='1'}
	ManualSamplingAck           : DINT;
	{attribute 'OPC.UA.DA':='1'}
	CleanedPartSamplingStatus   : DINT;
	{attribute 'OPC.UA.DA':='1'}
	CleanedPartSamplingAck      : DINT;
	{attribute 'OPC.UA.DA':='1'}
	LastSamplingQuantity        : DINT;
	{attribute 'OPC.UA.DA':='1'}
	LastSamplingAck             : DINT;
	{attribute 'OPC.UA.DA':='1'}
	PeriodicSamplingFrequency   : DINT;

END_VAR

// ---- GVLs/SerialComm.TcGVL
{attribute 'qualified_only'}
VAR_GLOBAL
		TxBuffer_1: COMbuffer;
		RxBuffer_1: COMbuffer;
END_VAR

// ---- GVLs/XTS/GVL_XTS.TcGVL
VAR_GLOBAL CONSTANT
	nNumberOfMovers		: INT:=31;
	nNumberOfStations	: INT:=35;

END_VAR

VAR_GLOBAL
	Mover : ARRAY[1..nNumberOfMovers] OF AXIS_REF;
	
	fbXTSEnvironment	 : FB_TcIoXtsEnvironment;
	CAGroup				 : AXES_GROUP_REF;
	DEVSTATE  AT %I*	: UINT;
	
END_VAR
VAR_GLOBAL PERSISTENT
	retain_1: BOOL;
	
	
// ALL MOVER STOP POSITIONS

	
	OP10A_STN_POSITION				:LREAL;
	OP10B_STN_POSITION				:lREAL;
	OP20_STN_POSITION               :lREAL;
    OP30_STN_POSITION               :lREAL;
	OP40_STN_POSITION               :LREAL;
	OP50_STN_POSITION               :lREAL;
	OP60_STN_POSITION               :lREAL;
	OP70_STN_POSITION               :lREAL;
	OP80_STN_POSITION               :lREAL;
	OP90_STN_POSITION               :lREAL;
	OP100_STN_POSITION              :lREAL;
	OP110_STN_POSITION              :lREAL;
	OP120_STN_POSITION              :lREAL;
	OP130_STN_POSITION              :lREAL;
	OP140_STN_POSITION              :lREAL;
	OP150_STN_POSITION              :lREAL;
	OP160_STN_POSITION              :LREAL;

																	  
																			 
						                                                   
                                                                      
                                                                      
																	   
   	END_VAR

// ---- POU1/Recipe_Values.TcGVL

VAR_GLOBAL PERSISTENT
	
//General
	Model_Dia					: STRING[80];
	Part_Number					: STRING[80];
	Body_Conductivity			: BOOL;
	Comp_Per_Bag 				: INT;
		
//OP10	
	OP10_Cam_Prog_Num			: INT;
	OP10_Robot_Prog_Num			: INT;
	OP10_Gripper_Pos			: REAL;
	
OP10_Bowl_freq_6_3				: REAL;
OP10_Conv_Fwd_Time_6_3			: INT;
OP10_Conv_Fwd_Speed_6_3			: INT;
OP10_Conv_Rev_Time_6_3			: INT;
OP10_Conv_Rev_Speed_6_3			: INT;
OP10_Hopper_ON_time_6_3			: INT;
OP10_Hopper_freq_6_3			: REAL;
OP10_Lnr_Trck_Dly_6_3			: REAL;

OP10_Bowl_freq_7_89				: REAL;	
OP10_Conv_Fwd_Time_7_89			: INT;
OP10_Conv_Fwd_Speed_7_89		: INT;
OP10_Conv_Rev_Time_7_89			: INT;
OP10_Conv_Rev_Speed_7_89		: INT;
OP10_Hopper_ON_time_7_89		: INT;
OP10_Hopper_freq_7_89			: REAL;
OP10_Lnr_Trck_Dly_7_89			: REAL;

//OP20
	OP20_Vert_Ser_Pos			: REAL;
	OP20_Oiling_Time			: INT;
	
OP20_Oiling_Range				: REAL;

//OP30
	OP30_Cam_Prog_Num			: INT;
	OP30_Grip_Wrk_Pos			: REAL;
	OP30_Vert_Ser_Pick_Pos		: REAL;
	OP30_Vert_Ser_Place_Pos		: REAL;	
	OP30_Hori_Ser_Pick_Pos		: REAL;
	OP30_Hori_Ser_Place_Pos		: REAL;		

//OP40
	OP40_Vert_Ser_Pos			: REAL;
	OP40_LVDT_Chck_Value		: REAL;

//OP40_LVDT_Tolerance				: REAL;

//OP50
	OP50_Cam_Prog_Num			: INT;
	OP50_Vert_Ser_Pick_Pos		: REAL;
	OP50_Vert_Ser_Place_Pos		: REAL;	
	OP50_Hori_Ser_Pick_Pos		: REAL;
	OP50_Hori_Ser_Place_Pos		: REAL;		

//OP60
	OP60_Vert_Ser_Pos			: REAL;
	OP60_LVDT_Chck_Value		: REAL;

//OP60_LVDT_Tolerance				: REAL;

//OP70
	OP70_Cam_Prog_Num			: INT;
	OP70_Grip_Wrk_Pos			: REAL;
	OP70_Vert_Ser_Pick_Pos		: REAL;
	OP70_Vert_Ser_Place_Pos		: REAL;	
	OP70_Hori_Ser_Pick_Pos		: REAL;
	OP70_Hori_Ser_Place_Pos		: REAL;		


//OP80
	OP80_Vert_Ser_Pos			: REAL;
	OP80_LVDT_Chck_Value		: REAL;

//OP80_LVDT_Tolerance				: REAL;

//OP90
	OP90_Cam_Prog_Num			: INT;
	OP90_Vert_Ser_Pick_Pos		: REAL;
	OP90_Vert_Ser_Place_Pos		: REAL;	
	OP90_Hori_Ser_Pick_Pos		: REAL;
	OP90_Hori_Ser_Place_Pos		: REAL;	

OP90_Bowl_freq_7_89				: REAL;	
OP90_Conv_Fwd_Time_7_89			: INT;
OP90_Conv_Fwd_Speed_7_89		: INT;
OP90_Conv_Rev_Time_7_89			: INT;
OP90_Conv_Rev_Speed_7_89		: INT;
OP90_Lnr_Trck_Dly_7_89			: REAL;

OP90_Bowl_freq_6_3				: REAL;	
OP90_Conv_Fwd_Time_6_3			: INT;
OP90_Conv_Fwd_Speed_6_3			: INT;
OP90_Conv_Rev_Time_6_3			: INT;
OP90_Conv_Rev_Speed_6_3			: INT;
OP90_Lnr_Trck_Dly_6_3			: REAL;

//OP110
	OP110_Vert_Ser_Pos			: REAL;
	OP110_Oiling_Time			: INT;
	
OP110_Oiling_Range				: REAL;

//OP120
	OP120_Cam_Prog_Num			: INT;

OP120_Bowl_freq 				: REAL;	
OP120_Conv_Fwd_Time 			: INT;
OP120_Conv_Fwd_Speed 			: INT;
OP120_Conv_Rev_Time 			: INT;
OP120_Conv_Rev_Speed 			: INT;
OP120_Lnr_Trck_Dly 				: REAL;
                            	
//OP130                     	
	OP130_Trq_value				: REAL;
	OP130_Vert_Ser_Pos			: REAL;
	                        	
//OP140                     	
	OP140_Vert_Ser_Pos			: REAL;
	                        	
OP140_Wiping_Cycle				: INT;
OP140_NOK_Retry_Cycle			: INT;
                            	
//OP150-A                   	
	OP150A_Cam_Prog_Num			: INT;
	                        	
//OP150-B                   	
	OP150B_Lsr_Mrk_Job_num		: INT;
	
//OP160
	OP160_Robo_Prog_Num			: INT;

END_VAR

// ---- POUs/GENERAL/GENERAL_VARIABLE.TcGVL
VAR_GLOBAL
	STATION_ENABLE_CONTROL				: BOOL;
	ManualMOde          :BOOL;
	OperationEnable     :BOOL;
	MODE_WORD			:INT;
	ALL_STN_IN_HOME		:BOOL;
	SAFE_TO_WORK		:BOOL; 
	START_PB			:BOOL;
	MODE_CHANGE_ACK		:BOOL;
	RESET_PB			:BOOL; //Mapped
	AUTO_SELECTED		:BOOL;
	MANUAL_SELECTED		:BOOL;
	STEP_SELECTED		:BOOL;
	AUTO_RUNNING		:BOOL;
	STEP_RUNNING		:BOOL;
	START_ENABLE		:BOOL;
	MACHINE_STOP		:BOOL;
	FB_MODE_BLOCK		:MODE_SELECTION_BLOCK1;
	ERROR_ACTIVE		:BOOL;
	IO_Page_Number		: INT;
	
	HMI_AutoMode   : BOOL;
	HMI_ManualMode : BOOL;
	HMI_StepMode   : BOOL;
	HMI_Reset	   : BOOL;
	
	HMI_Target_Count : DINT;
	HMI_Total_Count  : DINT;
	HMI_OK_Count	 : DINT;
	HMI_NOK_Count	 : DINT;
	
	All_Station_Dry_Run	: BOOL;
	
	Pulse_Block      : FB_SimClock;
	Servo_Enable     : BOOL;
    Servo_Safety     : BOOL;
    Servo_Reset      : BOOL;
//////********************************

    sNetID    : T_AmsNetID := '';
    bEnable   : BOOL;
    dwCycle   : DWORD(1..86400) := 5;
    dwOpt     : DWORD := 1;
    tTimeout  : TIME := DEFAULT_ADS_TIMEOUT;
	
	bValid     : BOOL;
    systemTime : TIMESTRUCT;
    tzID       : E_TimeZoneID := eTimeZoneID_Invalid;
	
    fbTime   : FB_LocalSystemTime := ( bEnable := TRUE, dwCycle := 1 );
    logTimer : TON := ( IN := TRUE, PT := T#10MS );	
	
	wYear	: WORD ;
	wMonth	: WORD ;
	wDate   : WORD ;
	wHour	: WORD ;
	wMinute : WORD ;
	wSecond : WORD ;
	wMillisec: WORD;	
//##############################		END_OF_CYCLE		##############################

		END_OF_CYCLE					: BOOL;


	
//################################		TOOL  CHANGE OVER 	#########################

		model_selected 					: INT;
END_VAR

VAR_GLOBAL PERSISTENT

		STN_BYPASS_ARAAY					: ARRAY[0..35] OF ARRAY[0..35]OF BOOL;
		STN_BYPASS_ARRAY_HMI				: ARRAY[0..35] OF BOOL;					
		ZERO_POS_XTS				        : LREAL :=0;
		XTS_POSITION						: ARRAY[2..35] OF LREAL;
		OP10A_BYPASS						: BOOL;
		OP10B_BYPASS		                : BOOL;
		OP20_BYPASS	                        : BOOL;
		OP30_BYPASS		                    : BOOL;
		OP40_BYPASS		                    : BOOL;
		OP50_BYPASS		                    : BOOL;
		OP60_BYPASS		                    : BOOL;
		OP70_BYPASS		                    : BOOL;
		OP80_BYPASS		                    : BOOL;
		OP90_BYPASS		                    : BOOL;
		OP110_BYPASS	                    : BOOL;
		OP120_BYPASS                        : BOOL;
		OP130_BYPASS                        : BOOL;
		OP140_P1_BYPASS                     : BOOL;
		OP140_P2_BYPASS                     : BOOL;
		OP140_P3_BYPASS                     : BOOL;
		OP150A_BYPASS                    	: BOOL;
		OP150B_BYPASS                    	: BOOL;
		OP150C_BYPASS                    	: BOOL;
		OP160_BYPASS                        : BOOL;
		Model								:STRING[80]:='6.3';
				
		OP10A_CURR_MOVER					: INT;
		OP10B_CURR_MOVER					: INT;		
		OP20_CURR_MOVER						: INT;
		OP30_CURR_MOVER						: INT;
		OP40_CURR_MOVER						: INT;
		OP50_CURR_MOVER						: INT;
		OP60_CURR_MOVER						: INT;
		OP70_CURR_MOVER						: INT;
		OP80_CURR_MOVER						: INT;		
		OP90_CURR_MOVER						: INT;	
		OP110_CURR_MOVER					: INT;
		OP120_CURR_MOVER					: INT;
		OP130_CURR_MOVER					: INT;
		OP140_P1_CURR_MVR					: INT;
		OP140_P2_CURR_MVR					: INT;
		OP140_P3_CURR_MVR					: INT;
//		OP150A_LH_CURR_MVR					: INT;
//		OP150A_RH_CURR_MVR					: INT;
//		OP150B_LH_CURR_MVR					: INT;
//		OP150B_RH_CURR_MVR					: INT;		
//		OP150C_LH_CURR_MVR					: INT;
//		OP150C_RH_CURR_MVR					: INT;		
//		OP160_CURR_MOVER					: INT;
END_VAR

// ---- POUs/IO_GVLs/Master3_IO.TcGVL

VAR_GLOBAL
	//port1
I90_RET_LH_GRIPR_CYL_CLSE_I1200_0              :BOOL;
I90_RET_LH_GRIPR_CYL_OPN_I1200_1               :BOOL;
I90_RET_RH_GRIPR_CYL_CLSE_I1200_2              :BOOL;
I90_RET_RH_GRIPR_CYL_OPN_I1200_3               :BOOL;
I90_POSTN_SLIDE_CYL_REV_I1200_4                :BOOL;
I90_POSTN_SLIDE_CYL_FWD_I1200_5                :BOOL;
I90_LH_MOVR_SUP_VERT_CYL_DWN_I1200_6           :BOOL;
I90_LH_MOVR_SUP_VERT_CYL_UP_I1200_7            :BOOL;
											  
I90_LH_MOVR_SUP_HORZ_CYL_REV_I1201_0           :BOOL;
I90_LH_MOVR_SUP_HORZ_CYL_FWD_I1201_1           :BOOL;
I90_RH_MOVR_SUP_VERT_CYL_DWN_I1201_2           :BOOL;
I90_RH_MOVR_SUP_VERT_CYL_UP_I1201_3            :BOOL;
I90_RH_MOVR_SUP_HORZ_CYL_REV_I1201_4           :BOOL;
I90_RH_MOVR_SUP_HORZ_CYL_FWD_I1201_5           :BOOL;
I90_SPARE_I1201_6                              :BOOL;
I90_SPARE_I1201_7                              :BOOL;

//port2
I90_LH1_REJ_SLIDE_REV_I1210_0                  :BOOL;
I90_LH1_REJ_SLIDE_FWD_I1210_1                  :BOOL;
I90_RH1_REJ_SLIDE_REV_I1210_2                  :BOOL;
I90_RH1_REJ_SLIDE_FWD_I1210_3                  :BOOL;
I90_LH2_REJ_SLIDE_REV_I1210_4                  :BOOL;
I90_LH2_REJ_SLIDE_FWD_I1210_5                  :BOOL;
I90_RH2_REJ_SLIDE_REV_I1210_6                  :BOOL;
I90_RH2_REJ_SLIDE_FWD_I1210_7                  :BOOL;
											   
I90_SPARE_I1211_0                              :BOOL;
I90_SPARE_I1211_1                              :BOOL;
I90_SPARE_I1211_2                              :BOOL;
I90_SPARE_I1211_3                              :BOOL;
I90_SPARE_I1211_4                              :BOOL;
I90_SPARE_I1211_5                              :BOOL;
I90_SPARE_I1211_6                              :BOOL;
I90_SPARE_I1211_7                              :BOOL;

//port3
I120_PUSH_CYL_REV_I1220_0                      :BOOL;
I120_PUSH_CYL_FWD_I1220_1                      :BOOL;
I120_LH_SING_CYL_REV_I1220_2                   :BOOL;
I120_LH_SING_CYL_FWD_I1220_3                   :BOOL;
I120_CAMERA_SLIDE_CYL_REV_I1220_4               :BOOL;
I120_CAMERA_SLIDE_CYL_FWD_I1220_5               :BOOL;
I120_SLAVE1_PRSN_PARK_TRAY_I1220_6             :BOOL;
I120_SLAVE2_PRSN_PARK_TRAY_I1220_7             :BOOL;
											   
